// TwinCAT 3 PLC project PLC_OPEN_DRIVE
// Title: PlcOpenDrive
// Author: D.Hauer
// ProjectVersion: 00.50.3
// Description: MotionControl Achs Controller für externe Ansteuerung; NCI implementation
// ProgramVersion: 3.1.4022.4
// libraries:
//   Tc2_EtherCAT, * (Beckhoff Automation GmbH)
//   Tc2_MC2, * (Beckhoff Automation GmbH)
//   Tc2_MC2_Camming, * (Beckhoff Automation GmbH)
//   Tc2_MC2_Drive, * (Beckhoff Automation GmbH)
//   Tc2_NC, * (Beckhoff Automation GmbH)
//   Tc2_NCI, * (Beckhoff Automation GmbH)
//   Tc2_PlcInterpolation, * (Beckhoff Automation GmbH)
//   Tc2_Standard, * (Beckhoff Automation GmbH)
//   Tc2_System, * (Beckhoff Automation GmbH)
//   Tc2_Utilities, * (Beckhoff Automation GmbH)
//   Tc3_Module, * (Beckhoff Automation GmbH)
// project tree:
//   DOC/ DOCUMENTATION.TcPOU
//   DUTs/AXIS_CONTROL/ e_AxisFunction.TcDUT, ST_AxisController.TcDUT, ST_CamIn.TcDUT, ST_MotionOptions.TcDUT, ST_DataLog.TcDUT, ST_GearIn.TcDUT, ST_GearInMultiMaster.TcDUT, ST_Homing.TcDUT, ST_NcParam.TcDUT, ST_AxisStatusCompact.TcDUT, ST_In.TcDUT, ST_Out.TcDUT
//   DUTs/MAPPING/ U_AXIS_CTRL.TcDUT, U_AXIS_GEAR_IN.TcDUT, U_AXIS_GEAR_IN_MULTIMASTER.TcDUT, U_AXIS_HOMING.TcDUT, U_AXIS_INFO.TcDUT, U_AXIS_MOTION_OPTIONS.TcDUT, U_AXIS_NC_PARAMETER.TcDUT, U_AXIS_STATE.TcDUT
//   DUTs/MESSAGE/ e_Device.TcDUT, E_MessageType.TcDUT, e_Subdevice.TcDUT, ST_Message.TcDUT
//   DUTs/NC_AXIS/ E_AxisEncoderType.TcDUT, ST_AxisName.TcDUT, ST_BoolParam.TcDUT, ST_GearInParams.TcDUT, ST_GetCamInfoParams.TcDUT, ST_HaltParams.TcDUT, ST_HaltPhasingParams.TcDUT, ST_HomeParams.TcDUT, ST_JogParams.TcDUT, ST_MoveAbsParams.TcDUT, ST_MoveVeloParams.TcDUT, ST_Param.TcDUT, ST_PhasingAbsParams.TcDUT, ST_PhasingRelParams.TcDUT, ST_ReadParamParams.TcDUT, ST_StopParams.TcDUT, ST_WriteParamParams.TcDUT
//   / GlobalTextList.TcGTLO, PlcTask.TcTTO, Visualisierungsmanager.TcVMO (not stored)
//   GVLs/ GVL_AXIS_CTRL.TcGVL
//   POUs/Functions/ f_Builder.TcPOU, f_DelBit64.TcPOU, f_FolderDate.TcPOU, f_GetBit64.TcPOU, f_Len.TcPOU, f_Setbit64.TcPOU
//   POUs/ MAIN.TcPOU, NCI.TcPOU, P_CopleyWorkAround.TcPOU
//   POUs/MAPPING/ MAPPING_in.TcPOU, MAPPING_out.TcPOU
//   POUs/MSG/ fb_WriteData.TcPOU, f_MessageSet.TcPOU, p_Data.TcPOU, Visualization.TcVIS
//   POUs/NCI/ e_Ctrl_NciCommand.TcDUT, e_NciChannelError.TcDUT, E_NCI_INTERPRETER_STATE.TcDUT, FB_Ctrl_NciChannel.TcPOU, FB_NciChannel.TcPOU, GVL_NCI.TcGVL, I_NciChannel.TcIO, I_Nci_Ctrl.TcIO, ST_3D_Group.TcDUT, ST_CTRL_NCI.TcDUT, ST_Ctrl_NciMFuncCycle.TcDUT, ST_Index_Group.TcDUT, ST_Interface_Group.TcDUT, ST_NciChannel_Ref.TcDUT, ST_R_Parameter.TcDUT, ST_STATE_NCI.TcDUT
//   POUs/NC_AXIS/ FB_McPtpAxis.TcPOU, I_McAxis.TcIO
//   POUs/_FunctionBlocks/cam/ FB_CamIn_empty.TcPOU, fb_Camming.TcPOU, fb_Camming_Empty.TcPOU, FB_CamOut_Empty.TcPOU
//   POUs/_FunctionBlocks/ FB_AxisController.TcPOU, fb_Blink.TcPOU, fb_LocalTime.TcPOU, fb_ResetSercos.TcPOU, FB_XenaxEtherCATHoming.TcPOU

CONFIGURATION PLC_OPEN_DRIVE
    RESOURCE PLC ON TwinCAT3
        TASK PlcTask(INTERVAL := T#1ms, PRIORITY := 20);
        PROGRAM MAPPING_in WITH PlcTask : MAPPING_in;
        PROGRAM MAIN WITH PlcTask : MAIN;
        PROGRAM NCI WITH PlcTask : NCI;
        PROGRAM MAPPING_out WITH PlcTask : MAPPING_out;
    END_RESOURCE
END_CONFIGURATION

// ---- DUTs/AXIS_CONTROL/e_AxisFunction.TcDUT
{attribute 'to_string'}
TYPE e_AxisFunction :
(
  AXIS_DISABLE,
  AXIS_IDLE := 1,
  AXIS_ENABLE := 10,
  AXIS_HOME,
  AXIS_MOVE_POS,
  AXIS_MOVE_VELO,
  AXIS_RESET,
  AXIS_HALT,
  AXIS_STOP,

  // TODO: test
  AXIS_MOVE_BUFFER := 20,
  AXIS_MOVE_BUFFER_VELO,
  AXIS_WRITE_BUFFER_MODE,


  AXIS_PARAMETER   := 30, // axis function for reading and writing parameter


  AXIS_GEAR_IN    := 50,
  AXIS_GEAR_OUT,
  AXIS_GEAR_IN_MULTIMASTER,

  AXIS_CAM_IN   := 60,
  AXIS_CAM_OUT,
  AXIS_CAM_INFO,

  AXIS_SS1_STOP   :=  99,
  AXIS_BUSY       := 100,
  AXIS_ACK        := 300,
  AXIS_DONE       := 1000,

  ERROR           := 9000
)UINT;
END_TYPE

// ---- DUTs/AXIS_CONTROL/ST_AxisController.TcDUT
{attribute 'pack_mode' := '2'}
TYPE ST_AxisController :
STRUCT
  ToPlc    : ST_In;
  FromPlc  : ST_Out;
END_STRUCT
END_TYPE

// ---- DUTs/AXIS_CONTROL/ST_CamIn.TcDUT
TYPE ST_CamIn :
STRUCT
  MasterOffset      : REAL; 
  SlaveOffset       : REAL; 
  MasterScaling     : REAL;
  SlaveScaling      : REAL;

{IF defined (CAM)}
  {info 'CAMMING active'}
  StartMode         : Tc2_MC2_Camming.MC_StartMode;
  CamTableID        : Tc2_MC2_Camming.MC_CAM_ID;
{ELSE}
  StartMode         : INT;
  CamTableID        : UDINT;
{END_IF}

END_STRUCT
END_TYPE

// ---- DUTs/AXIS_CONTROL/ST_MotionOptions.TcDUT
TYPE ST_MotionOptions :
STRUCT
  eBufferMode   : Tc2_MC2.MC_BufferMode;

END_STRUCT
END_TYPE

// ---- DUTs/AXIS_CONTROL/ST_DataLog.TcDUT
TYPE ST_DataLog :
STRUCT
  WorkOrder : WORD;
  Duration  : REAL; // [ms]
  Position  : REAL;
END_STRUCT
END_TYPE

// ---- DUTs/AXIS_CONTROL/ST_GearIn.TcDUT
{attribute 'pack_mode' := '2'}
TYPE ST_GearIn :
STRUCT
  RatioNumerator  : REAL := 1.0; 
  RatioDenominator: UINT := 1; 
  Acceleration    : REAL;
  Deceleration    : REAL;
  Jerk            : REAL;
END_STRUCT
END_TYPE

// ---- DUTs/AXIS_CONTROL/ST_GearInMultiMaster.TcDUT
{attribute 'pack_mode' := '2'}
TYPE ST_GearInMultiMaster :
STRUCT  
  byAxisIDMaster1  : BYTE; // AxisID of Master1
  byAxisIDMaster2  : BYTE; // AxisID of Master2
  byAxisIDMaster3  : BYTE; // AxisID of Master3
  byAxisIDMaster4  : BYTE; // AxisID of Master4
  GearRatio1       : REAL; 
  GearRatio2       : REAL; 
  GearRatio3       : REAL; 
  GearRatio4       : REAL; 
  Acceleration     : REAL;
  Deceleration     : REAL;
  Jerk             : REAL;  
END_STRUCT
END_TYPE

// ---- DUTs/AXIS_CONTROL/ST_Homing.TcDUT
TYPE ST_Homing :
STRUCT
  bExecute      : BIT;

  stHomingParam : ST_HomeParams;
END_STRUCT
END_TYPE

// ---- DUTs/AXIS_CONTROL/ST_NcParam.TcDUT
TYPE ST_NcParam :
STRUCT
  bRead           : BIT;
  bWrite          : BIT;
  bValid          : BIT;

  (* reserve for future use *)
  // TwinCAT fills up to byte alignement, the declarations are not neccessarily required
  // for ease of use placeholders are hidden from intelli sense
  {attribute 'hide'}
  b3 : BIT;
  {attribute 'hide'}
  b4 : BIT;
  {attribute 'hide'}
  b5 : BIT;
  {attribute 'hide'}
  b6 : BIT;
  {attribute 'hide'}
  b7 : BIT;
  {attribute 'hide'}
  by1 : BYTE;

  ParameterNumber : Tc2_MC2.MC_AxisParameter;
  rValueWrite     : REAL; // value to write
  rValueRead      : REAL; // value from NC (Bools are cast to real)
END_STRUCT
END_TYPE

// ---- DUTs/AXIS_CONTROL/ST_AxisStatusCompact.TcDUT
{attribute 'pack_mode' := '2'}
TYPE ST_AxisStatusCompact :
STRUCT

    Error                : BIT;  (* axis error state *)

    (* PLCopen motion control statemachine states: *)
    ErrorStop            : BIT;
    Disabled             : BIT;
    Stopping             : BIT;

    StandStill           : BIT;
    DiscreteMotion       : BIT;
    ContinuousMotion     : BIT; 
    SynchronizedMotion   : BIT;

    Homing               : BIT;

    (* additional status - (PLCopen definition)*)
    ConstantVelocity     : BIT; 
    Accelerating         : BIT;
    Decelerating         : BIT;

    (* Axis.NcToPlc.StateDWord *)
    Operational          : BIT; 
    ControlLoopClosed    : BIT; (* operational and position control active *)
    HasJob               : BIT; 
    HasBeenStopped       : BIT; 
    NewTargetPosition    : BIT; (* new target position commanded during move *)
    InPositionArea       : BIT; 
    InTargetPosition     : BIT; 
 
    Homed                : BIT; 
    HomingBusy           : BIT; 
    MotionCommandsLocked : BIT; (* stop 'n hold *)
    SoftLimitMinExceeded : BIT; (* reverse soft travel limit exceeded *)
    SoftLimitMaxExceeded : BIT; (* forward soft travel limit exceeded *)

    Moving               : BIT; 
    PositiveDirection    : BIT; 
    NegativeDirection    : BIT; 
    NotMoving            : BIT; 
    Compensating         : BIT; (* superposition - overlayed motion *)

    ExtSetPointGenEnabled: BIT; 
    ExternalLatchValid   : BIT; 
    CamDataQueued        : BIT; 
    CamTableQueued       : BIT; 
    CamScalingPending    : BIT; 
    CmdBuffered          : BIT; 
    PTPmode              : BIT; 
    DriveDeviceError     : BIT; 
    IoDataInvalid        : BIT; 

    (* Axis.NcToPlc.CoupleState *)
    Coupled              : BIT;

END_STRUCT
END_TYPE

// ---- DUTs/AXIS_CONTROL/ST_In.TcDUT
{attribute 'pack_mode' := '2'}
TYPE ST_In :
STRUCT


  bFastStop         : BIT;  // Fast stop function of NC with mapped input

  {attribute 'hide'}
  b1 : BIT; // hide bit; for future use
  {attribute 'hide'}
  b2 : BIT; // hide bit; for future use
  {attribute 'hide'}
  b3 : BIT; // hide bit; for future use
  {attribute 'hide'}
  b4 : BIT; // hide bit; for future use
  {attribute 'hide'}
  b5 : BIT; // hide bit; for future use
  {attribute 'hide'}
  b6 : BIT;
  {attribute 'hide'}
  b7 : BIT;

  byAxisFuncPara    : BYTE; // additional parameter for Axis Function; e.g. used for AxisIndex on GearIn

  uiAxisFunctionReq : e_AxisFunction; // selected function for axis 

  (* LREAL required by process *)
  rSetPos           : LREAL;
  rSetVelo          : LREAL;
  rOverride         : LREAL;
  rAcc              : LREAL;
  rDec              : LREAL;
  iDirection        : INT;

  {attribute 'hide'}
  w1 : ARRAY[1..3] OF WORD;

END_STRUCT
END_TYPE

// ---- DUTs/AXIS_CONTROL/ST_Out.TcDUT
{attribute 'pack_mode' := '2'}
TYPE ST_Out :
STRUCT

  bEnabled    : BIT; // Enabled: check if ControlLoop is closed and active
  bReferenced : BIT; // Axis homing bit
  bReady      : BIT; // enabled & NOT bError & no Axis Function requested
  bBusy       : BIT; // axis function requested or active
  bError      : BIT;
  bTimeout    : BIT; // for move cmds or switching drive on timeout
  bInTarget   : BIT; // ActPos = SetPos --> position check is done with configured window in NC
  bStandstill : BIT; // No Error and NOT moving

  byAxisFuncPara      : BYTE; // mirror for additional parameter for Axis Function; e.g. used for AxisIndex on GearIn
  uiAxisFunctionState : e_AxisFunction; // mirror the requested axis function; 
                                        // +  100 = function busy; 
                                        // + 1000 = function done; 
                                        // + 9000 = function error
  uiErrorId           : UDINT;

  rActPos             : LREAL;
  rActVelo            : LREAL;
  rPosDiff            : LREAL;

  rSetPos             : LREAL;

  // HAUD
  // 2023 04 05
  dwCoupleState       : DWORD;   // cyclic information about axis couple state

  {attribute 'hide'}
  w1 : ARRAY[1..4] OF WORD;
END_STRUCT
END_TYPE

// ---- DUTs/MAPPING/U_AXIS_CTRL.TcDUT
TYPE U_AXIS_CTRL :
UNION

  stCtrl              : ARRAY[1..GVL_AXIS_CTRL.gciMaxAxis] OF ST_In;

{IF defined (AXIS_MAP)}
  {info 'U_AXIS_CTRL mapping activated'}
  byCtrl    AT %I*    : ARRAY[1..GVL_AXIS_CTRL.gciMaxAxis] OF
                        ARRAY[1..SIZEOF(ST_In)] OF BYTE;
{ELSE}
  byCtrl              : ARRAY[1..GVL_AXIS_CTRL.gciMaxAxis] OF
                        ARRAY[1..SIZEOF(ST_In)] OF BYTE;
{END_IF}
END_UNION
END_TYPE

// ---- DUTs/MAPPING/U_AXIS_GEAR_IN.TcDUT
TYPE U_AXIS_GEAR_IN :
UNION

  stCtrl              : ARRAY[1..GVL_AXIS_CTRL.gciMaxAxis] OF ST_GearIn;

{IF defined (AXIS_MAP)}
  {info 'U_AXIS_GEAR_IN mapping activated'}
  byCtrl    AT %I*    : ARRAY[1..GVL_AXIS_CTRL.gciMaxAxis] OF
                        ARRAY[1..SIZEOF(ST_GearIn)] OF BYTE;
{ELSE}
  byCtrl              : ARRAY[1..GVL_AXIS_CTRL.gciMaxAxis] OF
                        ARRAY[1..SIZEOF(ST_GearIn)] OF BYTE;
{END_IF}
END_UNION
END_TYPE

// ---- DUTs/MAPPING/U_AXIS_GEAR_IN_MULTIMASTER.TcDUT
TYPE U_AXIS_GEAR_IN_MULTIMASTER :
UNION

  stCtrl              : ARRAY[1..GVL_AXIS_CTRL.gciMaxAxis] OF ST_GearInMultiMaster;

{IF defined (AXIS_MAP)}
  {info 'U_AXIS_GEAR_IN mapping activated'}
  byCtrl    AT %I*    : ARRAY[1..GVL_AXIS_CTRL.gciMaxAxis] OF
                        ARRAY[1..SIZEOF(ST_GearInMultiMaster)] OF BYTE;
{ELSE}
  byCtrl              : ARRAY[1..GVL_AXIS_CTRL.gciMaxAxis] OF
                        ARRAY[1..SIZEOF(ST_GearInMultiMaster)] OF BYTE;
{END_IF}
END_UNION
END_TYPE

// ---- DUTs/MAPPING/U_AXIS_HOMING.TcDUT
TYPE U_AXIS_HOMING :
UNION

  stCtrl              : ARRAY[1..GVL_AXIS_CTRL.gciMaxAxis] OF ST_Homing;

{IF defined (AXIS_MAP)}
  {info 'U_AXIS_HOMING mapping activated'}
  byCtrl    AT %I*    : ARRAY[1..GVL_AXIS_CTRL.gciMaxAxis] OF
                        ARRAY[1..SIZEOF(ST_Homing)] OF BYTE;
{ELSE}
  byCtrl              : ARRAY[1..GVL_AXIS_CTRL.gciMaxAxis] OF
                        ARRAY[1..SIZEOF(ST_Homing)] OF BYTE;
{END_IF}
END_UNION
END_TYPE

// ---- DUTs/MAPPING/U_AXIS_INFO.TcDUT
TYPE U_AXIS_INFO :
UNION

  stState             : ARRAY[1..GVL_AXIS_CTRL.gciMaxAxis] OF ST_AxisStatusCompact;

{IF defined (AXIS_MAP)}
  {info 'U_AXIS_INFO mapping activated'}
  byState  AT %Q*     : ARRAY[1..GVL_AXIS_CTRL.gciMaxAxis] OF
                        ARRAY[1..SIZEOF(ST_AxisStatusCompact)] OF BYTE;
{ELSE}
  byState             : ARRAY[1..GVL_AXIS_CTRL.gciMaxAxis] OF
                        ARRAY[1..SIZEOF(ST_AxisStatusCompact)] OF BYTE;
{END_IF}
END_UNION
END_TYPE

// ---- DUTs/MAPPING/U_AXIS_MOTION_OPTIONS.TcDUT
TYPE U_AXIS_MOTION_OPTIONS :
UNION

  stCtrl              : ARRAY[1..GVL_AXIS_CTRL.gciMaxAxis] OF ST_MotionOptions;

{IF defined (AXIS_MAP)}
  {info 'U_AXIS_MOTION_OPTIONS mapping activated'}
  byCtrl    AT %I*    : ARRAY[1..GVL_AXIS_CTRL.gciMaxAxis] OF
                        ARRAY[1..SIZEOF(ST_MotionOptions)] OF BYTE;
{ELSE}
  byCtrl              : ARRAY[1..GVL_AXIS_CTRL.gciMaxAxis] OF
                        ARRAY[1..SIZEOF(ST_MotionOptions)] OF BYTE;
{END_IF}
END_UNION
END_TYPE

// ---- DUTs/MAPPING/U_AXIS_NC_PARAMETER.TcDUT
TYPE U_AXIS_NC_PARAMETER :
UNION

  stState             : ARRAY[1..GVL_AXIS_CTRL.gciMaxAxis] OF ST_NcParam;

{IF defined (AXIS_MAP)}
  {info 'U_AXIS_NC_PARAM mapping activated'}
  byState   AT %Q*    : ARRAY[1..GVL_AXIS_CTRL.gciMaxAxis] OF
                        ARRAY[1..SIZEOF(ST_NcParam)] OF BYTE;
{ELSE}
  byState             : ARRAY[1..GVL_AXIS_CTRL.gciMaxAxis] OF
                        ARRAY[1..SIZEOF(ST_NcParam)] OF BYTE;
{END_IF}
END_UNION
END_TYPE

// ---- DUTs/MAPPING/U_AXIS_STATE.TcDUT
TYPE U_AXIS_STATE :
UNION

  stState             : ARRAY[1..GVL_AXIS_CTRL.gciMaxAxis] OF ST_Out;

{IF defined (AXIS_MAP)}
  {info 'U_AXIS_STATE mapping activated'}
  byState   AT %Q*    : ARRAY[1..GVL_AXIS_CTRL.gciMaxAxis] OF
                        ARRAY[1..SIZEOF(ST_Out)] OF BYTE;
{ELSE}
  byState             : ARRAY[1..GVL_AXIS_CTRL.gciMaxAxis] OF
                        ARRAY[1..SIZEOF(ST_Out)] OF BYTE;
{END_IF}
END_UNION
END_TYPE

// ---- DUTs/MESSAGE/e_Device.TcDUT
{attribute 'to_string'}
TYPE e_Device :
(
  General         := 0,

  // first NC Axis, all other Axis are incremented
  Axis            := 1000,

  // NCI channel control instance
  NciChannelCtrl  := 2000,

  // NCI channel
  NciChannel      := 3000,

  // message function blocks
  Data            := 10000
)DINT;
END_TYPE

// ---- DUTs/MESSAGE/E_MessageType.TcDUT
{attribute 'strict'}
{attribute 'to_string'}
TYPE E_MessageType :
(
  eMessageEmpty,
  eMessageInfo,
  eMessageWarn,
  eMessageError
)DINT;
END_TYPE

// ---- DUTs/MESSAGE/e_Subdevice.TcDUT
{attribute 'strict'}
{attribute 'to_string'}
TYPE e_Subdevice :
(
  // sub device for message system
  General := 0,
  // Motion Control FB Instances
  fbPower,
  fbReset,
  fbResetSercos,
  fbHalt,
  fbStop,
  fbHome,
  fbJog,
  fbMoveVelocity1,
  fbMoveVelocity2,
  fbMoveAbsolute1,
  fbMoveAbsolute2,
  fbMoveEndless,
  fbMovePtP,

  fbGearIn := 50,
  fbGearOut,
  fbGearInMultiMaster,

  fbCamIn := 60,
  fbCamOut,

  fbReadParameter := 100,
  fbReadBoolParameter,
  fbWriteParameter,
  fbWriteBoolParameter,

	fbBuildGroup := 200,
	fbClearGroup,
	fbLoadProg,
	fbResetItp,
	fbStartStopItp,
	fbEStopItp,
	fbStepOnAfterEStopItp,
	fbConfirmHskItp,
	fbDelDtgItp,
	fbNciFeedTablePreparation,
	fbNciFeedTable,
	fbReadLine,
  fbItpReadRParams,
  fbItpWriteRParams,

  Get_ItpState,
  Get_Error,

  AxisMode      := 1000,

  Ctrl_Nci_Cmd  := 2000
)DINT;
END_TYPE

// ---- DUTs/MESSAGE/ST_Message.TcDUT
TYPE ST_Message :
STRUCT
  eType         : e_MessageType;
  eDevice       : e_Device;
  eSubdevice    : e_SubDevice;
  {attribute 'displaymode':='hex'}
  iErrorNumber  : LINT;
  tTime         : STRING(24);
  sText         : STRING(256);
END_STRUCT
END_TYPE

// ---- DUTs/NC_AXIS/E_AxisEncoderType.TcDUT
{attribute 'to_string'}
TYPE E_AxisEncoderType :
(
  NoEncoder := 0,
  
  Simulation_Encoder,
  
  M3000_Enc,
  M31x0_M2000_Enc,
  MDP_511_Enc,
  MDP_500_501_Enc,
  MDP_510_Enc,
  KL30xx_Enc,
  SERCOS_EtherCAT_SoE_Pos,
  SERCOS_EtherCAT_SoE_Pos_Velo,
  Binary_Enc,
  M2510_Enc,
  FOX50_Enc                     := 12,
  AX2000_Lightbus               := 14,
  Provi_DriveMC_Simodrive_611U,
  Universal_Encoder_varBitmask,
  NC_Backplane,
  spec_CANopen_Typ,
  MDP_513_DS402,
  AX2xx_B900,
  KL5151_Encoder                := 21,
  IP5209_Encoder                := 24,
  KL2531_KL2541_Encoder,
  KL2532_KL2542_Encoder,
  Time_Base_Encoder,
  TCom_Encoder_SoftDrive
)UDINT;
END_TYPE

// ---- DUTs/NC_AXIS/ST_AxisName.TcDUT
TYPE ST_AxisName :
STRUCT
  sName     : STRING(31);
  bValid    : BOOL;
END_STRUCT
END_TYPE

// ---- DUTs/NC_AXIS/ST_BoolParam.TcDUT
TYPE ST_BoolParam :
STRUCT
  bValue      : BOOL;
  bValid      : BOOL;
  bWriteToNc  : BOOL;
END_STRUCT
END_TYPE

// ---- DUTs/NC_AXIS/ST_GearInParams.TcDUT
TYPE ST_GearInParams :
STRUCT
  Enable        : BOOL;
  GearRatio     : LREAL;
  GearRatio2    : LREAL;
  GearRatio3    : LREAL;
  GearRatio4    : LREAL;
  Acceleration  : LREAL;
  Deceleration  : LREAL;
  Jerk          : LREAL;
  Options       : Tc2_MC2.ST_GearInMultiMasterOptions;
END_STRUCT
END_TYPE

// ---- DUTs/NC_AXIS/ST_GetCamInfoParams.TcDUT
TYPE ST_GetCamInfoParams :
STRUCT
  AtMasterPosition  : BOOL;
  MasterPosition    : LREAL;
END_STRUCT
END_TYPE

// ---- DUTs/NC_AXIS/ST_HaltParams.TcDUT
TYPE ST_HaltParams :
STRUCT
  Deceleration  : LREAL;
  Jerk          : LREAL;
  BufferMode    : Tc2_MC2.MC_BufferMode;
END_STRUCT
END_TYPE

// ---- DUTs/NC_AXIS/ST_HaltPhasingParams.TcDUT
TYPE ST_HaltPhasingParams :
STRUCT
  Deceleration  : LREAL;
  Jerk          : LREAL;
END_STRUCT
END_TYPE

// ---- DUTs/NC_AXIS/ST_HomeParams.TcDUT
TYPE ST_HomeParams :
STRUCT
  Position              : LREAL;
  HomingMode            : Tc2_MC2.MC_HomingMode;
  Options               : Tc2_MC2.ST_HomingOptions;
  InvertHomeSensor      : BIT := FALSE;   //Set to true, if the home sensor is normally closed.
  SimulateHomeSensor    : BIT := FALSE;   //Set to true, if the axis should be homed on encoder index only. The homing methode 'hardware sync' must be used then.
  UseLimitMin           : BIT := TRUE;    //Set to false, if there is no negative limit sensor.
  InvertLimitMin        : BIT := FALSE;   //Set to true, if the negative limit sensor is normally closed.
  HomeOnLimitMin        : BIT := FALSE;   //Set to true, if the negative limit sensor should be used for homing. 
  UseLimitMax           : BIT := TRUE;    //Set to false, if there is no positive limit sensor.
  InvertLimitMax        : BIT := FALSE;   //Set to true, if the positive limit sensor is normally closed.
  HomeOnLimitMax        : BIT := FALSE;   //Set to true, if the positive limit sensor should be used for homing. 
  
  // It is not allowed to use more than 1 of the 3 switches: SimulateHomeSensor, HomeOnLimitMin, HomeOnLimitMax
  
END_STRUCT
END_TYPE

// ---- DUTs/NC_AXIS/ST_JogParams.TcDUT
TYPE ST_JogParams :
STRUCT
  JogForward    : BOOL;
  JogBackwards  : BOOL;
  Mode          : Tc2_MC2.E_JogMode;
  Position      : LREAL;
  Velocity      : LREAL;
  Acceleration  : LREAL;
  Deceleration  : LREAL;
  Jerk          : LREAL;
END_STRUCT
END_TYPE

// ---- DUTs/NC_AXIS/ST_MoveAbsParams.TcDUT
TYPE ST_MoveAbsParams :
STRUCT
	Position		: LREAL;
	Velocity		: LREAL;
	Acceleration	: LREAL;
	Deceleration	: LREAL;
	Jerk			: LREAL;
	BufferMode		: Tc2_MC2.MC_BufferMode;
END_STRUCT
END_TYPE

// ---- DUTs/NC_AXIS/ST_MoveVeloParams.TcDUT
TYPE ST_MoveVeloParams :
STRUCT
  Velocity      : LREAL;
  Acceleration  : LREAL;
  Deceleration  : LREAL;
  Jerk          : LREAL;
  Direction     : Tc2_MC2.MC_Direction := MC_Positive_Direction;
  BufferMode    : Tc2_MC2.MC_BufferMode;
END_STRUCT
END_TYPE

// ---- DUTs/NC_AXIS/ST_Param.TcDUT
TYPE ST_Param :
STRUCT
  fValue    : LREAL;
  bValid    : BOOL;
  bWriteToNc  : BOOL;
END_STRUCT
END_TYPE

// ---- DUTs/NC_AXIS/ST_PhasingAbsParams.TcDUT
TYPE ST_PhasingAbsParams :
STRUCT
	PhaseShift		: LREAL;
	Velocity		: LREAL;
	Acceleration	: LREAL;
	Deceleration	: LREAL;
	Jerk			: LREAL;
END_STRUCT
END_TYPE

// ---- DUTs/NC_AXIS/ST_PhasingRelParams.TcDUT
TYPE ST_PhasingRelParams :
STRUCT
	PhaseShift		: LREAL;
	Velocity		: LREAL;
	Acceleration	: LREAL;
	Deceleration	: LREAL;
	Jerk			: LREAL;
END_STRUCT
END_TYPE

// ---- DUTs/NC_AXIS/ST_ReadParamParams.TcDUT
TYPE ST_ReadParamParams :
STRUCT
	ParameterNumber	: Tc2_MC2.MC_AxisParameter;
END_STRUCT
END_TYPE

// ---- DUTs/NC_AXIS/ST_StopParams.TcDUT
TYPE ST_StopParams :
STRUCT
	Deceleration	: LREAL;
	Jerk			: LREAL;
END_STRUCT
END_TYPE

// ---- DUTs/NC_AXIS/ST_WriteParamParams.TcDUT
TYPE ST_WriteParamParams :
STRUCT
  ParameterNumber : Tc2_MC2.MC_AxisParameter;
  Value           : LREAL;
END_STRUCT
END_TYPE

// ---- POUs/NCI/e_Ctrl_NciCommand.TcDUT
{attribute 'qualified_only'}
{attribute 'to_string'}
TYPE e_Ctrl_NciCommand :
(
  NO_NCI            := -10,
  NO_AXIS_GROUP     := -2,
  NO_AXIS_INDEX     := -1,
  NO_INIT,
  INIT,
  IDLE,
  RESET,
  LOAD_PROG,
  FEED_TABLE,
  BUILD_GROUP,
  CLEAR_GROUP,

  START         := 10,
  STOP,
  STO_STOP,
  RESTART_STEP_ON,

  M_FUNC_QUIT   := 20,

  READ_R_PARA   := 30,
  WRITE_R_PARA  := 40,

  CMD_BUSY      := 100,
  CMD_DONE      := 1000,
  CMD_ERROR     := 9000
)DINT;
END_TYPE

// ---- POUs/NCI/e_NciChannelError.TcDUT
{attribute 'qualified_only'}
{attribute 'strict'}
TYPE e_NciChannelError :
(
  e_Null,
  e_InvalidReference_ChannelRef,
  e_AxisConfigurationMismatch_McAxis,
  e_AxisConfigurationMismatch_AuxAxis


);
END_TYPE

// ---- POUs/NCI/E_NCI_INTERPRETER_STATE.TcDUT
// Interpreter state, see also library tc2_nci.Global_Variables.NCI_INTERPRETER_xxx
//  Date    Name  Version   Remarks
//  2016/09/29  FJK   1.0     1st Version
{attribute -'to_string'}
TYPE E_NCI_INTERPRETER_STATE :
(
  NCI_INTERPRETER_INITFAILED := 0,
  NCI_INTERPRETER_IDLE := 1,
  NCI_INTERPRETER_READY := 2,
  NCI_INTERPRETER_STARTED := 3,
  NCI_INTERPRETER_SCANNING := 4,
  NCI_INTERPRETER_RUNNING := 5,
  NCI_INTERPRETER_STAY_RUNNING := 6,
  NCI_INTERPRETER_WRITETABLE := 7,
  NCI_INTERPRETER_SEARCHLINE := 8,
  NCI_INTERPRETER_END := 9,
  NCI_INTERPRETER_SINGLESTOP := 10, 
  NCI_INTERPRETER_ABORTING := 11,
  NCI_INTERPRETER_ABORTED := 12,
  NCI_INTERPRETER_FAULT := 13,
  NCI_INTERPRETER_RESET := 14,
  NCI_INTERPRETER_STOP := 15,
  NCI_INTERPRETER_WAITFUNC := 16,
  NCI_INTERPRETER_FLUSHBUFFERS := 17
) DWORD;    //Basis-Datentyp
END_TYPE

// ---- POUs/NCI/ST_3D_Group.TcDUT
{attribute 'pack_mode' := '2'}
TYPE ST_3D_Group :
STRUCT
  nXAxisId    : UDINT := 1;
  nYAxisId    : UDINT := 2;
  nZAxisId    : UDINT := 3;
  nQ1AxisId   : UDINT;
  nQ2AxisId   : UDINT;
  nQ3AxisId   : UDINT;
  nQ4AxisId   : UDINT;
  nQ5AxisId   : UDINT;
END_STRUCT
END_TYPE

// ---- POUs/NCI/ST_CTRL_NCI.TcDUT
{attribute 'pack_mode' := '2'}
TYPE ST_CTRL_NCI :
STRUCT
  eCmd        : e_Ctrl_NciCommand := e_Ctrl_NciCommand.INIT;
  rOverride   : REAL := 47.11;

END_STRUCT
END_TYPE

// ---- POUs/NCI/ST_Ctrl_NciMFuncCycle.TcDUT
{attribute 'pack_mode' := '2'}
TYPE ST_Ctrl_NciMFuncCycle :
STRUCT
  FastMFuncMask   : ARRAY [1..5] OF DWORD;
  HskMFuncNo      : UINT;
  HskMFuncReq     : WORD;
  HFuncValue      : UDINT; 
END_STRUCT
END_TYPE

// ---- POUs/NCI/ST_Index_Group.TcDUT
{attribute 'pack_mode' := '2'}
TYPE ST_Index_Group :
STRUCT
  nXAxisIdx     : UDINT := 1;
  nYAxisIdx     : UDINT := 2;
  nZAxisIdx     : UDINT := 3;

  nQ1AxisIdx    : UDINT;
  nQ2AxisIdx    : UDINT;
  nQ3AxisIdx    : UDINT;
  nQ4AxisIdx    : UDINT;
  nQ5AxisIdx    : UDINT;
END_STRUCT
END_TYPE

// ---- POUs/NCI/ST_Interface_Group.TcDUT
{attribute 'pack_mode' := '2'}
TYPE ST_Interface_Group :
STRUCT
  I_Idx_XAxis     : I_McAxis;
  I_Idx_YAxis     : I_McAxis;
  I_Idx_ZAxis     : I_McAxis;

  I_Idx_Q1Axis    : I_McAxis;
  I_Idx_Q2Axis    : I_McAxis;
  I_Idx_Q3Axis    : I_McAxis;
  I_Idx_Q4Axis    : I_McAxis;
  I_Idx_Q5Axis    : I_McAxis;
END_STRUCT
END_TYPE

// ---- POUs/NCI/ST_NciChannel_Ref.TcDUT
TYPE ST_NciChannel_Ref :
STRUCT
  NcToPlc AT %I*: NcToPlc_NciChannel_Ref;   //  Externer Datentyp!
  PlcToNc AT %Q*: PlcToNc_NciChannel_Ref;   //  Externer Datentyp!
END_STRUCT
END_TYPE

// ---- POUs/NCI/ST_R_Parameter.TcDUT
{attribute 'pack_mode' := '2'}
TYPE ST_R_Parameter :
STRUCT
{IF defined (AXIS_MAP)}
  {info 'NCI channel mapping for test'}
  _nStart        AT %I* : DINT;
  _nCount        AT %I* : DINT;
  _rRParamsWrite AT %I* : ARRAY[0..GVL_NCI.cRParamCount] OF LREAL;
  _rRParamsRead  AT %Q* : ARRAY[0..GVL_NCI.cRParamCount] OF LREAL;
{ELSE}
  _nStart               : DINT := 901;
  _nCount               : DINT :=   4;
  _rRParamsWrite        : ARRAY[0..GVL_NCI.cRParamCount] OF LREAL := [11.11, 22.22, 33.33, 456.22];
  _rRParamsRead         : ARRAY[0..GVL_NCI.cRParamCount] OF LREAL;
{END_IF}
END_STRUCT
END_TYPE

// ---- POUs/NCI/ST_STATE_NCI.TcDUT
{attribute 'pack_mode' := '2'}
TYPE ST_STATE_NCI :
STRUCT
  eState        : e_Ctrl_NciCommand; // eCmd with offsets for busy and done

  bMFuncReq     : BIT;  // M function request is active from channel

  nMFunc        : WORD; // number of active M function

  nItpState     : UINT; 
                         (*  Interpreter Operation State:
                            0  = Init failed
                            1  = Idle
                            2  = Ready
                            3  = Started
                            4  = Scanning
                            5  = Running
                            6  = Stay running
                            7  = Write table
                            8  = Search line
                            9  = End
                            10 = Single Step
                            11 = Aborting
                            12 = Aborted
                            13 = Fault
                            14 = Reset
                            15 = Stop
                            16 = Wait function
                            17 = Flush buffers
                          *) 

  rAxisOverride : REAL; // active override in cyclic NCI interface

END_STRUCT
END_TYPE

// ---- GVLs/GVL_AXIS_CTRL.TcGVL
{attribute 'qualified_only'}
VAR_GLOBAL CONSTANT

{IF defined (WIN)}
  {info 'WIN folders'}
  gcsLogDir         : STRING := 'C:\TwinCAT\#MsgFiles\';
{ELSE}
  {info 'BSD folders'}
  gcsLogDir         : STRING := '/usr/local/etc/TwinCAT/#MsgFiles/';
{END_IF}

  gcsLogFile        : STRING := 'Msg_PlcOpenDrive_';

  gciMaxMessage     : INT := 200; // max entry in message list
  gciMaxAxis        : INT :=  3;

{IF defined (CAM)}
  {info 'camming active'}
  cCam                  : BOOL := TRUE;
{ELSE}
  {info 'camming NOT active'}
  cCam                  : BOOL := FALSE;
{END_IF}

  
//V 00.07
//04.11.2021
//HauD
// GearIn, GearOut added

// V 00.08
//24.03.2022
//HauD
// simple ptp movement with only one instance of MC functionblock
// file writing for logging now globally enable/disable
// intern message list is always used
// ref in property deleted
// axis pointer is used


// V 00.09
// 25.03.2022
// HAUD
// parameter handling changed
// NULL initialization of methods implemented

// V 00.10 - V 00.11
// 29.03.2022
// HAUD
// TEST

// V 00.12
// 29.03.2022
// HAUD
// Merge TEST and server version
// Visu page for message diag
// OP state before ADS READ on NC Axis
// INIT logging at startup
// enum to_string with use of 4024 compiler

// V 00.13
// 14.04.2022
// CamIn and CamOut added
// Changed Compiler Version to 3.1.4024.0. This is needed to enable conditional pragmas

// V 00.14
// 03.06.2022
// GearInMultiMaster added

// V 00.15
// 29.06.2022
// HAUD
// defines deleted, defines in code do not work, therefore all defines for camming deleted
// stop method in FB_McPtPAxis added.

// V00.16
// 30.06..2022
// HAUD
// FB_AxisController, code refactoring
//    Axis function states are now calling corresponding actions to improve readability
// SS1 stop with static check (SEL)

// V00.17
// 18.07.2022
// HAUD
// CAM_OUT now with FB check instead of mapping check

// V00.18
// 19.07.2022
// Axis startup, changes according to test
// ADS communication to AxisName changed, ADS Err 1796

// V00.19
// 27.07.2022
// HAUD
// Axis startup expanded to Encodertype for automatic Sercos selection
// fb_AxisController.bSercosAxis changed from input to output var
// CamOut checked with logging for couple state

// V00.20
// 27.07.2022
// HAUD
// Axis startup AdsRead.ERR automatic re-startup

// V00.21
// 06.10.2022
// HAUD
// test case for MOVE_VELO; HALT
// Halt() with standstill check
// MOVE_VELO, fbMoveEndless.Position feed check
// AXIS_HALT, standstill control with timeout and RESET
// AXIS_MOVE_BUFFER_VELO, two instances changing velocity during function execution, if required velo is reached, done OR keep function alive and change to velo2 and wait for done


// V00.22
// 13.10.2022
// HAUD
// AXIS_HALT standstill check changed to NotMoving

// V00.23
// 14.10.2022
// HAUD
// AXIS_MOVE_VELO - chsnged to MC_Velocity; Ctrl.iDirection is evaluated, 1 - positive; 3 - negative

// V00.24
// 15.10.2022
// HAUD
// code revision from testing
// Compiler def TEST      - TwinSAFE Alias device muted
// Compiler def AXIS_MAP  - cyclic mapping ST_AxisController
// Compiler def WIN       - windows file names for logging

// V00.25
// 15.10.2022
// HAUD
// Compiler def CAM      - contitional activation of camming lib
// MC_Camming lib now optional

// V00.26
// 16.10.2022
// HAUD
// cam folder missing, added by push
// property of MC2_Camming.lib is set to optional
// Compiler def:  - TEST      [forces SafetyOK internally]
//                - AXIS_MAP  [ST_AxisController will be mapped variable --> connection to second TEST_PLC]
//                - WIN       [windows file names are used]
//                - CAM       [MC2_Camming.lib is active --> if entry is not present, empty FBs are used]

// V00.27
// 19.10.2022
// HAUD
// R/W of axis parameter now possible without safety bit from Alias Device

// V00.28
// 20.10.2022
// HAUD
// GearOut and Disable are available during safety off.

// V00.30
// 23.10.2022
// HAUD
// NCI implementation of for basic use with g-Code files

// V00.32
// 25.10.2022
// HAUD
// consistent Datatypes for NCI define

// V00.33
// 25.10.2022
// HAUD
// NCI() call added to TaskReference
// NCI() works the ADS interface
// cyclic interface for NCI channels as global data structs
// plausibility checks

// V00.34
// 25.10.2022
// HAUD
// compiler defines test

// V00.35
// 25.10.2022
// HAUD
// BUG fb_AxisController.bSS1 state bereinigt

// V00.36
// 25.10.2022
// HAUD
// defines for test cases with mapping to extern plc
// 

// V00.37
// 25.10.2022
// HAUD
// defines for test cases with mapping to extern plc
// properties in fb_Ctrl_NciChannel are now using fb Instance of FB_NciChannel
// R Parameter window limited to 10

// V00.38
// 25.10.2022
// HAUD
// testing

// V00.39
// 31.10.2022
// HAUD
// quit of M function now on cyclic interface
// new member in ST_STATE_NCI  .ItpState - Interpreter state from cyclic NCI channel interfacwe 

// V00.40
// 02.11.2022
// HAUD
// testing

// V00.41
// 18.01.2023
// - BufferMode switch for e_AxisFunction.AXIS_MOVE_BUFFER and AXIS_MOVE_BUFFER_VELO

// V00.42
// HAUD
// 14.03.2023
// CAM_OUT check changed to strict eval

// V00.43
// HAUD
// 17.03.2023
// MC_BufferModes, additional error check in FB_McPtpAxis added (MoveAbsolute 1&2)

// V00.44
// HAUD
// 17.03.2023
// code review for missing stState.uiErrorId information to extern

// V00.45
// HAUD
// 27.03.2023
// debug for missing stState.uiErrorId information to extern
//
// 31.03.2023
// Axis_Cam_Out; ignore fb_CamOut error, retry if still coupled

// V00.46
// HAUD
// 05.04.2023
// Axis_Cam_Out; ignore axis function if not coupled
// fbAxis.pAxisRef^.NcToPlc.CoupleState added to ST_OUT

// V00.47
// HAUD
// 27.04.2023
// draft for redesign Camming lib implementation
// fb_CamIn_V2 replaces fb_CamIn

// V00.48 new branch on git server
// HAUD
// 26.05.2023
// ST_In; ST_Out change REAL --> LREAL

// V00.48.01
// HAUD
// 17.10.2023
// more than 100 Axis declared in project --> ADS handles can not be created for all axis, StartUp FB_McPtpAxis stopps with error, manual reset required --> changed to closer monitoring and retry
// FB_McPtpAxis.StartupError    - added if ADS Read error, StartUp error state wait for Reset
// FB_McPtpAxis.ErrorReset      - added StartUp error state reset (restarts StartUp state machine)
// FB_AxisController.Axis_Init  - state machine is checked for fbAxis.StartUpError, automatic axis reset and retry

// V00.50.1
// HAUD
// 19.10.2023
// CAMMING implementation with table manipulation
// redesign for modular use --> FB_AxisController does not host camming lib
// interface implementation for downward compatibility

// V00.48.93
// HAUD
// 15.02.2024
// Buffered moves with additional info on ST_Out.rSetPos

// V00.50.2
// HAUD
// 07.03.2024
// merge changes from field V 00.48.95
// buffered move
// message handling

// V00.50.3
// HAUD
// 11.03.2024
// AXIS_MAP pragma through dedicated PRG (in/out)



  Version           : STRING := 'V 00.50.3';
END_VAR
VAR_GLOBAL

  gfbAxisController : ARRAY[1..gciMaxAxis] OF FB_AxisController;  // cyclic interface for accepting and executing orders
  gstAxisControl    : ARRAY[1..gciMaxAxis] OF ST_AxisController;  // structure for cyclic interface


  gstAxisParam                  : ARRAY[1..gciMaxAxis] OF ST_NcParam;         // R/W struct for a single parameter
  gstHomeParam                  : ARRAY[1..gciMaxAxis] OF ST_HomeParams;      // homing parameter for each axis

  gstAxisCamParam               : ARRAY[1..gciMaxAxis] OF ST_CamIn;
  gstAxisGearParam              : ARRAY[1..gciMaxAxis] OF ST_GearIn;
  gstAxisGearMultiMasterParam   : ARRAY[1..gciMaxAxis] OF ST_GearInMultiMaster;

  gstMotionOptions              : ARRAY[1..gciMaxAxis] OF ST_MotionOptions;

  // diag data
  gbyAxisIdxGearIn              : ARRAY[1..gciMaxAxis]      OF BYTE; // diag for Axis gear in
  
  gbyAxisIdxGearInMultiMaster   : ARRAY[1..gciMaxAxis,1..4] OF BYTE; // diag for Axis gear in multi master
  
  gbyAxisIdxCamIn               : ARRAY[1..gciMaxAxis]      OF BYTE; // diag for Axis cam in

  gatMessages       : ARRAY[1..gciMaxMessage] OF ST_Message;
  giMsgIndex        : INT := 1;
  giErrorIndex      : INT := 0;

  gfbLocalTime      : fb_LocalTime;
  gdtLocalTime      : DT;
  gsLocalTime       : STRING;

{IF defined (AXIS_MAP)}
  {info 'TEST ST_AxisController'}
  gbEnableLogging   : BOOL := TRUE;
{ELSE}
  gbEnableLogging   : BOOL;
{END_IF}
END_VAR

// ---- POUs/NCI/GVL_NCI.TcGVL
{attribute 'qualified_only'}
VAR_GLOBAL CONSTANT
  cPathSteps            : UINT    := 5;  //Path-Steps[0]:Velo, [1]:X, [2]:Y, [3]:Z
  cMcAxisCount          : UINT    := 8;
  cAuxAxisCount         : UINT    := 8;
  cRParamCount          : UINT    := 10;

  cNciSpec              : STRING  := 'NCI_Spec_Ch_';

  cMaxNciCh             : INT     :=  1;

{IF defined (NCI)}
  {info 'NCI channel active'}
  cNci                  : BOOL := TRUE;
{ELSE}
  {info 'NCI channel NOT active'}
  cNci                  : BOOL := FALSE;
{END_IF}


{IF defined (WIN)}
  {info 'WIN folders'}
  cNciDir              : STRING   := 'C:\TwinCAT\Mc\Nci\';
{ELSE}
  {info 'BSD folders'}
  cNciDir              : STRING   := '/usr/local/etc/TwinCAT/Mc/Nci/';
{END_IF}
END_VAR
VAR_GLOBAL

{IF defined (AXIS_MAP)}
  {info 'NCI channel mapping for test'}
  gstAxisIndex      AT %I*    : ARRAY[1..cMaxNciCh] OF ST_Index_Group;  // index of gstAxisCtontrl[]
  gstAxisConfig     AT %I*    : ARRAY[1..cMaxNciCh] OF ST_3D_Group;     // NC Axis Id to build NCI group

  gstChannelCtrl    AT %I*    : ARRAY[1..cMaxNciCh] OF ST_CTRL_NCI;
  gstChannelState   AT %Q*    : ARRAY[1..cMaxNciCh] OF ST_STATE_NCI;

  gsProgName        AT %I*    : ARRAY[1..cMaxNciCh] OF STRING(255);
  gsProgNameActive  AT %Q*    : ARRAY[1..cMaxNciCh] OF STRING(255);
{ELSE}

  // ADS R/W data:
  gstAxisIndex                : ARRAY[1..cMaxNciCh] OF ST_Index_Group;  // index of gstAxisCtontrl[]
  gstAxisConfig               : ARRAY[1..cMaxNciCh] OF ST_3D_Group;     // NC Axis Id to build NCI group

  gstChannelCtrl              : ARRAY[1..cMaxNciCh] OF ST_CTRL_NCI;
  gstChannelState             : ARRAY[1..cMaxNciCh] OF ST_STATE_NCI;

  gsProgName                  : ARRAY[1..cMaxNciCh] OF STRING(255):= ['/usr/local/etc/TwinCAT/Mc/Nci/Test_GST.nc'];
  gsProgNameActive            : ARRAY[1..cMaxNciCh] OF STRING(255);
{END_IF}

  gstRParameter               : ARRAY[1..cMaxNciCh] OF ST_R_Parameter;

{IF defined (NCI)}
  gfbNciCtrl            : ARRAY[1..cMaxNciCh] OF FB_Ctrl_NciChannel;
{ELSE}
  gfbNciCtrl            : ARRAY[1..cMaxNciCh] OF I_Nci_Ctrl;
{END_IF}
END_VAR

// ---- POUs/NCI/I_NciChannel.TcIO
INTERFACE I_NciChannel

(*
===============================================================
Implementation of Tc2_NCI.CfgBuildExt3DGroup

  Builds complete NCI-Group with all configured axes
===============================================================
*)
METHOD BuildGroup : HRESULT
VAR_INPUT
  Execute: BOOL;
END_VAR
END_METHOD

(*
===============================================================
NCI-Group configured axes structure
===============================================================
*)
PROPERTY CfgAxes : Tc2_NCI.NCI_EXT3DGROUP
SET
END_SET
END_PROPERTY

(*
===============================================================
Implementation of Tc2_NCI.CfgReconfigGroup

  remove all axes from NCI-Group
===============================================================
*)
METHOD ClearGroup : HRESULT
VAR_INPUT
  Execute: BOOL;
END_VAR
END_METHOD

METHOD ConfirmHSK : HRESULT
VAR_INPUT
  Execute: BOOL;
END_VAR
END_METHOD

(*
===============================================================
Implementation of Tc2_NCI.ItpDelDtgEx

  DelDTG ( delete distance to go ) wird aus dem NC Programm satzweise aktiviert. 
  Dieses Kommando ermöglicht es, aus der SPS ( TcNci.lib ItpDelDtgEx) den Restweg der aktuellen Geometrie zu löschen. 
  D.h. trifft das Kommando während der Abarbeitung des Satzes ein so wird mit den üblichen Verzögerungsrampen die Bewegung angehalten. 
  Anschließend wird mit dem nächsten Satz im NC Programm fortgefahren.
  Falls das SPS-Kommando nicht während der Ausführung eines Satzes mit angewähltem Restweglöschen eintrifft, wird dieses mit einer Fehlermeldung beantwortet.
  Das Restweglöschen bewirkt immer einen impliziten Dekodierstop, d.h. es erfolgt am Satzende immer ein Genauhalt.
===============================================================
*)
METHOD DelDTG : HRESULT
VAR_INPUT
  Execute: BOOL;
END_VAR
END_METHOD

PROPERTY Error : BOOL
GET
END_GET
END_PROPERTY

METHOD Error_Get : BOOL
END_METHOD

(*
===============================================================
Implementation of Tc2_NCI.ItpEStopEx
===============================================================
*)
METHOD EStop : HRESULT
VAR_INPUT
  Execute: BOOL;
END_VAR
END_METHOD

METHOD GetChannelOverride : real
VAR_INPUT
END_VAR
END_METHOD

METHOD GetItpState : uint
VAR_INPUT
END_VAR
END_METHOD

PROPERTY HSK : BOOL
GET
END_GET
END_PROPERTY

PROPERTY I_AuxAxis : ARRAY[1..GVL_NCI.cAuxAxisCount] OF I_McAxis
SET
END_SET
END_PROPERTY

PROPERTY I_McAxis : array[1..GVL_NCI.cMcAxisCount] of I_McAxis
SET
END_SET
END_PROPERTY

PROPERTY ItpAxes : Tc2_NCI.NCI_EXT3DGROUP
GET
END_GET
END_PROPERTY

(*
===============================================================
Implementation of Tc2_NCI.ItpResetEx2
===============================================================
*)
METHOD ItpReset : HRESULT
VAR_INPUT
  Execute: BOOL;
END_VAR
END_METHOD

METHOD LoadProg : HRESULT
VAR_INPUT
  Execute: BOOL;
END_VAR
END_METHOD

PROPERTY MFunc : INT
GET
END_GET
END_PROPERTY

PROPERTY Override : LREAL
GET
END_GET
SET
END_SET
END_PROPERTY

PROPERTY PathVelo : LREAL
GET
END_GET
END_PROPERTY

PROPERTY pNciChannelRef : POINTER TO ST_NciChannel_Ref
GET
END_GET
END_PROPERTY

PROPERTY Prog : STRING(255)
GET
END_GET
SET
END_SET
END_PROPERTY

(*
===============================================================
Implementation of Tc2_System.ADSREADEX

  reads actual interpreter G-Code Line
===============================================================
*)
METHOD ReadLine : HRESULT
VAR_INPUT
  Execute: BOOL;
END_VAR
//Read G-Code actual Line
VAR_OUTPUT
  ActProgLine: STRING(100);
END_VAR
END_METHOD

(*
===============================================================
Implementation of Tc2_NCI.ItpReadRParamsEx

  read R-Parameter(s) from NCI
===============================================================
*)
METHOD ReadRParams : HRESULT
VAR_INPUT
  Execute :BOOL;
  Addr    :POINTER TO LREAL;  //Adresse der Zielvariablen der zu lesenden Daten. 
        //Dabei werden die Daten direkt ab der angegebenen Adresse von der NC beschrieben  
        //D.h. nIndex ist nicht als Offset zu pAddr zu sehen. Die Daten befinden sich z.B. 
        //in einem Array vom Typ LREAL, das vom Anwender definiert werden muss.
  Index   :DINT;
  Count   :DINT;
END_VAR
END_METHOD

(*
===============================================================
Implementation of Tc2_NCI.ItpStartStopEx

  Start Interpreter
===============================================================
*)
METHOD StartStop : HRESULT
VAR_INPUT
  Start: BOOL;
  Stop: BOOL;
END_VAR
END_METHOD

(*
===============================================================
Implementation of Tc2_NCI.ItpStopOnAfterEStopEx
===============================================================
*)
METHOD StepOnAfterEStop : HRESULT
VAR_INPUT
  Execute: BOOL;
END_VAR
END_METHOD

(*
===============================================================
Implementation of Tc2_NCI.ItpWriteRParamsEx

  write R-Parameter(s) to NCI
===============================================================
*)
METHOD WriteRParams : HRESULT
VAR_INPUT
  Execute :BOOL;
  Addr    :POINTER TO LREAL;  //Adresse der Zielvariablen der Daten. 
        //Dabei werden die Daten direkt ab der angegebenen Adresse von der NC beschrieben  
        //D.h. nIndex ist nicht als Offset zu pAddr zu sehen. Die Daten befinden sich z.B. 
        //in einem Array vom Typ LREAL, das vom Anwender definiert werden muss.
  Index   :DINT;
  Count   :DINT;
END_VAR
END_METHOD

END_INTERFACE

// ---- POUs/NCI/I_Nci_Ctrl.TcIO
INTERFACE I_Nci_Ctrl

PROPERTY ChnId : udint
GET
END_GET
END_PROPERTY

METHOD Cycle
VAR_INPUT
END_VAR
END_METHOD

PROPERTY eCmd : e_Ctrl_NciCommand
GET
END_GET
SET
END_SET
END_PROPERTY

PROPERTY eState : e_Ctrl_NciCommand
GET
END_GET
SET
END_SET
END_PROPERTY

PROPERTY GroupAxisConfig : ST_3D_Group
GET
END_GET
SET
END_SET
END_PROPERTY

PROPERTY I_AuxAxis : array[1..GVL_NCI.cAuxAxisCount] of I_McAxis
GET
END_GET
SET
END_SET
END_PROPERTY

PROPERTY I_McAxis : array[1..GVL_NCI.cMcAxisCount] of I_McAxis
GET
END_GET
SET
END_SET
END_PROPERTY

PROPERTY I_NcChannel : I_NciChannel
GET
END_GET
END_PROPERTY

PROPERTY M_FuncReq : word
GET
END_GET
END_PROPERTY

PROPERTY NcProg : string(255)
GET
END_GET
SET
END_SET
END_PROPERTY

PROPERTY R_Param_Read : ARRAY [0..GVL_NCI.cRParamCount] OF lreal
GET
END_GET
SET
END_SET
END_PROPERTY

PROPERTY R_Param_Write : ARRAY [0..GVL_NCI.cRParamCount] OF lreal
GET
END_GET
SET
END_SET
END_PROPERTY

PROPERTY R_ParamCount : DINT
GET
END_GET
SET
END_SET
END_PROPERTY

PROPERTY R_ParamIndex : DINT
GET
END_GET
SET
END_SET
END_PROPERTY

PROPERTY sCmd : string
GET
END_GET
SET
END_SET
END_PROPERTY

END_INTERFACE

// ---- POUs/NC_AXIS/I_McAxis.TcIO
INTERFACE I_McAxis

PROPERTY pAxisRef : pointer to AXIS_REF
GET
END_GET
END_PROPERTY

PROPERTY Position : LREAL
GET
END_GET
END_PROPERTY

END_INTERFACE

// ---- POUs/MAPPING/MAPPING_in.TcPOU
PROGRAM MAPPING_in
VAR CONSTANT
{IF defined (AXIS_MAP)}
  {info 'MAPPING_in - ACTIVE'}
  bBypassMapping    : BOOL  := FALSE;
{ELSE}
  bBypassMapping    : BOOL  := TRUE;
{END_IF}
END_VAR
VAR
  AxisCTrl              : U_AXIS_CTRL;
  AxisMotionOptions     : U_AXIS_MOTION_OPTIONS;

  AxisGearInData        : U_AXIS_GEAR_IN;
  AxisGearInMultiMaster : U_AXIS_GEAR_IN_MULTIMASTER;
  AxisHoming            : U_AXIS_HOMING;
  AxisParameterWrt      : U_AXIS_NC_PARAMETER;

  nAxis                 : INT;
END_VAR

IF bBypassMapping THEN RETURN; END_IF


FOR nAxis := 1 TO GVL_AXIS_CTRL.gciMaxAxis
DO
  memcpy(ADR(GVL_AXIS_CTRL.gstAxisControl[nAxis].ToPlc),  ADR(AxisCtrl.stCtrl[nAxis]),          SIZEOF(ST_In));
  memcpy(ADR(GVL_AXIS_CTRL.gstMotionOptions[nAxis]),      ADR(AxisMotionOptions.stCtrl[nAxis]), SIZEOF(ST_MotionOptions));
  memcpy(ADR(GVL_AXIS_CTRL.gstAxisGearParam[nAxis]),      ADR(AxisGearInData.stCtrl[nAxis]),    SIZEOF(ST_GearIn));
  memcpy(ADR(GVL_AXIS_CTRL.gstHomeParam[nAxis]),          ADR(AxisHoming.stCtrl[nAxis]),        SIZEOF(ST_HomeParams));

  GVL_AXIS_CTRL.gstAxisParam[nAxis].bRead             := AxisParameterWrt.stState[nAxis].bRead;
  GVL_AXIS_CTRL.gstAxisParam[nAxis].bWrite            := AxisParameterWrt.stState[nAxis].bWrite;
  GVL_AXIS_CTRL.gstAxisParam[nAxis].ParameterNumber   := AxisParameterWrt.stState[nAxis].ParameterNumber;
  GVL_AXIS_CTRL.gstAxisParam[nAxis].rValueWrite       := AxisParameterWrt.stState[nAxis].rValueWrite;
END_FOR

END_PROGRAM

// ---- POUs/MAIN.TcPOU
PROGRAM MAIN
VAR
	uiFrm0_State				AT %I* : UINT;
	uiFrm0_WcState			AT %I* : UINT;
	uiFrm0_InputToggle	AT %I* : UINT;
	uiSlaveCount				AT %I* : UINT;
	uiDevState					AT %I* : UINT;

{IF defined (TEST)}
  {info 'TEST'}
	bSafety_OK					       : BOOL := TRUE;
{ELSE}
	bSafety_OK					AT %I* : BOOL; // Input for TwinSAFE signal for SS1 stop
{END_IF}

	aOut	AT %Q* : BOOL;
	bTic				 : BOOL;
	diCounter		 : DINT;
	imod				 : INT := 10;

	szAxisCtrl, 
	szAxisCtrlPlc, 
	szAxisCtrlC, 
	szNcParam,
	szHomeParam	: UINT;
	iAxisIndex	: INT := 1;
	i						: INT;

	rtrigWriteFile		: R_TRIG;
  tonWriteFile      : TON;
  tWriteFile        : time := t#5s;
END_VAR

// Local time; used for timestamps
GVL_AXIS_CTRL.gfbLocalTime(sLocalTime=> GVL_AXIS_CTRL.gsLocalTime, dtLocalTime=> GVL_AXIS_CTRL.gdtLocalTime);


diCounter := diCounter + 1;

// tic for ADS notification
IF (diCounter MOD imod = 0)
THEN
	bTic          := NOT bTic;
	aOut          := NOT aOut;
END_IF

szAxisCtrl      := SIZEOF(GVL_AXIS_CTRL.gstAxisControl[iAxisIndex]);
szAxisCtrlPlc   := SIZEOF(GVL_AXIS_CTRL.gstAxisControl[iAxisIndex].ToPlc);
szAxisCtrlC     := SIZEOF(GVL_AXIS_CTRL.gstAxisControl[iAxisIndex].FromPlc);
szNcParam       := SIZEOF(GVL_AXIS_CTRL.gstAxisParam[iAxisIndex]);
szHomeParam     := SIZEOF(GVL_AXIS_CTRL.gstHomeParam[iAxisIndex]);

FOR i := 1 TO GVL_AXIS_CTRL.gciMaxAxis
DO
  CASE GVL_AXIS_CTRL.gstAxisControl[i].ToPlc.uiAxisFunctionReq 
  OF
    //-----------------------------------------------------------------------------------------------------------------
    // GearIn
    //-----------------------------------------------------------------------------------------------------------------
    e_AxisFunction.AXIS_GEAR_IN:

      IF(GVL_AXIS_CTRL.gstAxisControl[i].ToPlc.byAxisFuncPara > 0) AND
        (GVL_AXIS_CTRL.gstAxisControl[i].ToPlc.byAxisFuncPara <= GVL_AXIS_CTRL.gciMaxAxis)
      THEN
        // copy index to diag array
        GVL_AXIS_CTRL.gbyAxisIdxGearIn[i]                       := GVL_AXIS_CTRL.gstAxisControl[i].ToPlc.byAxisFuncPara; // FuncParam for GEAR_IN carries array index of master axis
        GVL_AXIS_CTRL.gfbAxisController[i].MasterAxis1          := GVL_AXIS_CTRL.gfbAxisController[GVL_AXIS_CTRL.gbyAxisIdxGearIn[i]].fbAxis.pAxisRef;
        GVL_AXIS_CTRL.gfbAxisController[i].stGear               := GVL_AXIS_CTRL.gstAxisGearParam[i];
        GVL_AXIS_CTRL.gstAxisControl[i].FromPlc.byAxisFuncPara  := GVL_AXIS_CTRL.gbyAxisIdxGearIn[i];
      END_IF


    //-----------------------------------------------------------------------------------------------------------------
    // GearInMultimaster
    //-----------------------------------------------------------------------------------------------------------------
    e_AxisFunction.AXIS_GEAR_IN_MULTIMASTER:

      // Master 1
      IF(GVL_AXIS_CTRL.gstAxisGearMultiMasterParam[i].byAxisIDMaster1 > 0) AND
        (GVL_AXIS_CTRL.gstAxisGearMultiMasterParam[i].byAxisIDMaster1 <= GVL_AXIS_CTRL.gciMaxAxis) 
      THEN
        GVL_AXIS_CTRL.gbyAxisIdxGearInMultiMaster[i,1]          := GVL_AXIS_CTRL.gstAxisGearMultiMasterParam[i].byAxisIDMaster1;
        GVL_AXIS_CTRL.gfbAxisController[i].MasterAxis1          := GVL_AXIS_CTRL.gfbAxisController[GVL_AXIS_CTRL.gstAxisGearMultiMasterParam[i].byAxisIDMaster1].fbAxis.pAxisRef;
      ELSE
        GVL_AXIS_CTRL.gbyAxisIdxGearInMultiMaster[i,1]          := 0;
        GVL_AXIS_CTRL.gfbAxisController[i].MasterAxis1          := 0;
      END_IF

      // Master 2
      IF(GVL_AXIS_CTRL.gstAxisGearMultiMasterParam[i].byAxisIDMaster2 > 0) AND
        (GVL_AXIS_CTRL.gstAxisGearMultiMasterParam[i].byAxisIDMaster2 <= GVL_AXIS_CTRL.gciMaxAxis)	  
      THEN
        GVL_AXIS_CTRL.gbyAxisIdxGearInMultiMaster[i,2]          := GVL_AXIS_CTRL.gstAxisGearMultiMasterParam[i].byAxisIDMaster2;
        GVL_AXIS_CTRL.gfbAxisController[i].MasterAxis2          := GVL_AXIS_CTRL.gfbAxisController[GVL_AXIS_CTRL.gstAxisGearMultiMasterParam[i].byAxisIDMaster2].fbAxis.pAxisRef;
      ELSE
        GVL_AXIS_CTRL.gbyAxisIdxGearInMultiMaster[i,2]          := 0;
        GVL_AXIS_CTRL.gfbAxisController[i].MasterAxis2          := 0;
      END_IF 

      // Master 3
      IF(GVL_AXIS_CTRL.gstAxisGearMultiMasterParam[i].byAxisIDMaster3 > 0) AND
       (GVL_AXIS_CTRL.gstAxisGearMultiMasterParam[i].byAxisIDMaster3 <= GVL_AXIS_CTRL.gciMaxAxis)
      THEN
        GVL_AXIS_CTRL.gbyAxisIdxGearInMultiMaster[i,3]          := GVL_AXIS_CTRL.gstAxisGearMultiMasterParam[i].byAxisIDMaster3;
        GVL_AXIS_CTRL.gfbAxisController[i].MasterAxis3          := GVL_AXIS_CTRL.gfbAxisController[GVL_AXIS_CTRL.gstAxisGearMultiMasterParam[i].byAxisIDMaster3].fbAxis.pAxisRef;
      ELSE
        GVL_AXIS_CTRL.gbyAxisIdxGearInMultiMaster[i,3]          := 0;
        GVL_AXIS_CTRL.gfbAxisController[i].MasterAxis3          := 0;
      END_IF

      // Master 4	 
      IF(GVL_AXIS_CTRL.gstAxisGearMultiMasterParam[i].byAxisIDMaster4 >= 0) AND
        (GVL_AXIS_CTRL.gstAxisGearMultiMasterParam[i].byAxisIDMaster4 <= GVL_AXIS_CTRL.gciMaxAxis)
      THEN
        GVL_AXIS_CTRL.gbyAxisIdxGearInMultiMaster[i,4]          := GVL_AXIS_CTRL.gstAxisGearMultiMasterParam[i].byAxisIDMaster4;
        GVL_AXIS_CTRL.gfbAxisController[i].MasterAxis4          := GVL_AXIS_CTRL.gfbAxisController[GVL_AXIS_CTRL.gstAxisGearMultiMasterParam[i].byAxisIDMaster4].fbAxis.pAxisRef;
      ELSE
        GVL_AXIS_CTRL.gbyAxisIdxGearInMultiMaster[i,4]          := 0;
        GVL_AXIS_CTRL.gfbAxisController[i].MasterAxis4          := 0;
      END_IF

      GVL_AXIS_CTRL.gfbAxisController[i].stGearMultiMaster      := GVL_AXIS_CTRL.gstAxisGearMultiMasterParam[i];


    //-----------------------------------------------------------------------------------------------------------------
    // CamIn
    //-----------------------------------------------------------------------------------------------------------------
    e_AxisFunction.AXIS_CAM_IN:

      IF(GVL_AXIS_CTRL.gstAxisControl[i].ToPlc.byAxisFuncPara > 0) AND
        (GVL_AXIS_CTRL.gstAxisControl[i].ToPlc.byAxisFuncPara <= GVL_AXIS_CTRL.gciMaxAxis)
      THEN
      // copy index to diag array
        GVL_AXIS_CTRL.gbyAxisIdxCamIn[i]                        := GVL_AXIS_CTRL.gstAxisControl[i].ToPlc.byAxisFuncPara; // FuncParam carries array index of master axis
      // assign master axis
        GVL_AXIS_CTRL.gfbAxisController[i].MasterAxis1          := GVL_AXIS_CTRL.gfbAxisController[GVL_AXIS_CTRL.gbyAxisIdxCamIn[i]].fbAxis.pAxisRef;
      // assign CAM parameters
        GVL_AXIS_CTRL.gfbAxisController[i].stCam                := GVL_AXIS_CTRL.gstAxisCamParam[i];
      // copy index to FromPLC structure 
        GVL_AXIS_CTRL.gstAxisControl[i].FromPlc.byAxisFuncPara  := GVL_AXIS_CTRL.gbyAxisIdxCamIn[i];
      END_IF


	
  ELSE  
    GVL_AXIS_CTRL.gbyAxisIdxGearIn[i]                           := 0;

    GVL_AXIS_CTRL.gbyAxisIdxGearInMultiMaster[i,1]              := 0;
    GVL_AXIS_CTRL.gbyAxisIdxGearInMultiMaster[i,2]              := 0;
    GVL_AXIS_CTRL.gbyAxisIdxGearInMultiMaster[i,3]              := 0;
    GVL_AXIS_CTRL.gbyAxisIdxGearInMultiMaster[i,4]              := 0;

    GVL_AXIS_CTRL.gbyAxisIdxCamIn[i]                            := 0;
    GVL_AXIS_CTRL.gfbAxisController[i].MasterAxis1              := 0;
  END_CASE


  //-----------------------------------------------------------------------------------------------------------------
  // Axis cyclic call
  //-----------------------------------------------------------------------------------------------------------------
	GVL_AXIS_CTRL.gfbAxisController[i](	stCtrl	                  := GVL_AXIS_CTRL.gstAxisControl[i].ToPlc,   // global struct to write on 

                                      bSS1						          := bSafety_OK, 
                                      stHomingOptions	          := GVL_AXIS_CTRL.gstHomeParam[i], 
                                      stNcParameter		          := GVL_AXIS_CTRL.gstAxisParam[i],
                                      stMotionOptions           := GVL_AXIS_CTRL.gstMotionOptions[i],

                                      stState					          => GVL_AXIS_CTRL.gstAxisControl[i].FromPlc  // global struct to read from
                                     );   
END_FOR

tonWriteFile(IN := TRUE, PT := tWriteFile);

IF tonWriteFile.Q
THEN
  p_Data.bWriteFile := TRUE;
  tonWriteFile(IN:=FALSE);
END_IF  

//-----------------------------------------------------------------------------------------------------------------
// write message list to file
//-----------------------------------------------------------------------------------------------------------------
p_Data(pList			:= ADR(GVL_AXIS_CTRL.gatMessages),
			 pLocalTime := ADR(GVL_AXIS_CTRL.gdtLocalTime), 
			 bBusy=> );



IF p_Data.bWriteFile AND
   p_Data.bBusy
THEN
  p_Data.bWriteFile := FALSE;
END_IF

P_CopleyWorkAround();

END_PROGRAM

// ---- POUs/MSG/p_Data.TcPOU
PROGRAM p_Data
VAR_INPUT
	bPowerFail		: BOOL;
	bWriteFile		: BOOL;
	bReset				: BOOL;
	pList					: POINTER TO ARRAY[1..GVL_AXIS_CTRL.gciMaxMessage] OF ST_Message;
	pLocalTime		: POINTER TO DT; 
END_VAR
VAR_OUTPUT
	bBusy					: BOOL;
	VisuList		  : ARRAY[1..GVL_AXIS_CTRL.gciMaxMessage] OF ST_Message;
END_VAR
VAR
	diStep 				: DINT;

	rtrigReset		: Tc2_Standard.R_TRIG;
	aWriteList		: ARRAY[1..GVL_AXIS_CTRL.gciMaxMessage] OF ST_Message;
	sWriteData		: STRING(32767);
	sNewLine			: STRING := '$N';
	sTab					: STRING := '$T';
	iCount, 
	iStart, 
	iEnd					: INT;

	fbWrite				: fb_WriteData;
	fbCreateDir		: Tc2_System.FB_CreateDir;
	sTmp          : STRING(256);
	sFilename			: STRING(256);
	sFolderDate		: STRING;
	bFileCreated	: BOOL;

  ivis          : INT;
END_VAR
VAR CONSTANT
	MSG_WRITE_COUNT	: INT := 10;
END_VAR

(* pointer check *)
IF NOT (pList <> 0) OR
	 NOT (pLocalTime <> 0)
THEN
	RETURN;
END_IF

IF (f_FolderDate(pLocalTime) <> sFolderDate)
THEN
	bFileCreated := FALSE;
END_IF


rtrigReset(CLK:= bReset);
IF rtrigReset.Q
THEN
	bReset := FALSE;
	diStep := 0;
END_IF


CASE diStep OF
	0:
		bBusy := FALSE;
    IF bWriteFile
    THEN
      diStep := 5;
		ELSIF (GVL_AXIS_CTRL.giMsgIndex >= MSG_WRITE_COUNT) OR
			     bPowerFail
		THEN
      diStep := 5;
	END_IF
END_CASE
CASE diStep OF
  5:
			memcpy(ADR(aWriteList), pList, SIZEOF(aWriteList));
			memset(pList, 0, SIZEOF(aWriteList));

			bBusy                             := TRUE;
			iStart 	                          := 1;
			iEnd 		                          := SEL((GVL_AXIS_CTRL.giMsgIndex > GVL_AXIS_CTRL.gciMaxMessage),
                                                GVL_AXIS_CTRL.giMsgIndex,
                                                GVL_AXIS_CTRL.gciMaxMessage);

			GVL_AXIS_CTRL.giMsgIndex          := 1;

			fbWrite.bExecute                  := FALSE;

			IF NOT bFileCreated
			THEN
        IF (GVL_AXIS_CTRL.giErrorIndex > 0)
        THEN
          GVL_AXIS_CTRL.giErrorIndex    := 0;
				  diStep                        := 10;
        ELSE
          diStep                        := 250;
        END_IF
			ELSE
        GVL_AXIS_CTRL.giErrorIndex      := 0;
				diStep := 200;
			END_IF
END_CASE
CASE diStep OF
	10:
		fbCreateDir.sPathName := left(GVL_AXIS_CTRL.gcsLogDir,len(GVL_AXIS_CTRL.gcsLogDir)-1);
		fbCreateDir.bExecute  := FALSE;
		diStep := 20;

	20:
		(* create root folder *)
		fbCreateDir.bExecute	:= TRUE;
		IF fbCreateDir.bBusy
		THEN
			diStep := 30;
		END_IF

	30:
		IF NOT fbCreateDir.bBusy
		THEN
			sFolderDate := f_FolderDate(pLocalTime);
			fbCreateDir.sPathName := concat(GVL_AXIS_CTRL.gcsLogDir, sFolderDate);
			fbCreateDir.bExecute  := FALSE;
			diStep := 40;
		END_IF

	40:
		(* create active folder *)
		fbCreateDir.bExecute	:= TRUE;
		IF fbCreateDir.bBusy
		THEN
			diStep := 50;
		END_IF

	50:
		IF NOT fbCreateDir.bBusy
		THEN
			fbCreateDir.bExecute  := FALSE;
			// build complete file path
			sTmp := concat(concat(GVL_AXIS_CTRL.gcsLogFile, sFolderDate),'.txt');
			sTmp := concat('\', sTmp);
			sFilename := concat(fbCreateDir.sPathName, sTmp);
			bFileCreated := TRUE;
			diStep := 200;
		END_IF

END_CASE
CASE diStep OF
	200:
		memset(ADR(sWriteData),0,SIZEOF(sWriteData));
		iCount := iStart;
		diStep := 220;

	220:
		IF aWriteList[iCount].eType > 0
		THEN
      IF (aWriteList[iCount].eType > E_MessageType.eMessageInfo) OR
          GVL_AXIS_CTRL.gbEnableLogging
      THEN
        sTmp := TO_STRING(aWriteList[iCount].eType);
        sTmp := Tc2_Standard.CONCAT(sTmp, sTab);
        sTmp := Tc2_Standard.CONCAT(sTmp, aWriteList[iCount].tTime);
        sTmp := Tc2_Standard.CONCAT(sTmp, sTab);
        sTmp := Tc2_Standard.CONCAT(sTmp, Device_To_String(aWriteList[iCount].eDevice));
        sTmp := Tc2_Standard.CONCAT(sTmp, sTab);
        sTmp := Tc2_Standard.CONCAT(sTmp, TO_STRING(aWriteList[iCount].eSubdevice));
        sTmp := Tc2_Standard.CONCAT(sTmp, sTab);
        sTmp := Tc2_Standard.CONCAT(sTmp, TO_STRING(aWriteList[iCount].iErrorNumber));
        sTmp := Tc2_Standard.CONCAT(sTmp, sTab);
        sTmp := Tc2_Standard.CONCAT(sTmp, aWriteList[iCount].sText);
        sTmp := Tc2_Standard.CONCAT(sTmp, sNewLine);
        f_Builder(ADR(sTmp), ADR(sWriteData), len(sTmp));
      END_IF
		END_IF
		iCount := iCount + 1;
		diStep := 225;

	225:
		IF iCount > iEnd
		THEN
			IF (len(sWriteData) > 0)
			THEN
				diStep := 230;
			ELSE
				diStep := 250;
			END_IF
		ELSE
			diStep := 220;
		END_IF


	230:
		fbWrite.bExecute 	:= TRUE;
		IF fbWrite.bBusy
		THEN
			diStep := 240;
		END_IF

	240:
		IF NOT fbWrite.bBusy
		THEN
			fbWrite.bExecute := FALSE;
			diStep := 250;
		END_IF

	250:
		IF NOT bWriteFile
		THEN
			diStep := 0;
		END_IF
END_CASE

fbWrite(
	bExecute:= , 
	sFileName:= sFilename, 
	psData:= ADR(sWriteData), 
	bBusy=> , 
	bDone=> , 
	bError=> );

fbCreateDir(
	sNetId:= , 
	sPathName:=, 
	ePath:= , 
	bExecute:= , 
	tTimeout:= , 
	bBusy=> , 
	bError=> , 
	nErrId=> );

// copy list for visu
FOR ivis := 1 TO GVL_AXIS_CTRL.giMsgIndex
DO
  VisuList[ivis] := pList^[ivis];
END_FOR

METHOD Device_to_String : string
VAR_INPUT
  eMsgDevice    : e_Device;
END_VAR
VAR
  // first NC Axis, all other Axis are incremented
  nmodAxis            : DINT := 1000;

  // first NCI channel control instance
  nmodNciChannelCtrl  : DINT := 2000;

  // NCI channel
  nmodNciChannel      : DINT := 3000;

  // message function blocks
  nmodData            : DINT := 10000;

  sId                 : STRING := '_ID_';
  nId                 : DINT;
END_VAR

IF (eMsgDevice <= nmodAxis)
THEN
  // general case with no added indices
  Device_to_String := TO_STRING(eMsgDevice);
ELSE

  IF (eMsgDevice > nModData)
  THEN
    nId := eMsgDevice MOD nmodData;
    sId := concat(sId, TO_STRING(nId));
 
    Device_to_String := concat(TO_STRING(e_device.Data), sId);

  ELSIF (eMsgDevice > nmodNciChannel)
  THEN
    nId := eMsgDevice MOD nmodNciChannel;
    sId := concat(sId, TO_STRING(nId));
 
    Device_to_String := concat(TO_STRING(e_device.NciChannel), sId);

  ELSIF (eMsgDevice > nmodNciChannelCtrl)
  THEN
    nId := eMsgDevice MOD nmodNciChannelCtrl;
    sId := concat(sId, TO_STRING(nId));
 
    Device_to_String := concat(TO_STRING(e_device.NciChannelCtrl), sId);

  ELSIF (eMsgDevice > nmodAxis)
  THEN
    nId := eMsgDevice MOD nmodAxis;
    sId := concat(sId, TO_STRING(nId));
 
    Device_to_String := concat(TO_STRING(e_device.Axis), sId);
  ELSE
    Device_to_String := TO_STRING(eMsgDevice);
  END_IF
END_IF
END_METHOD

END_PROGRAM

// ---- POUs/MSG/fb_WriteData.TcPOU
FUNCTION_BLOCK fb_WriteData
VAR_INPUT
	bExecute		: BOOL;
	sFileName		: Tc2_System.T_MaxString; (* filename and ending *)
	psData			: POINTER TO STRING(32767);
END_VAR
VAR_OUTPUT
	bBusy				: BOOL;
	bDone				: BOOL;
	bError			: BOOL;
END_VAR
VAR
	diStep			: DINT;
	udiCounter	: UDINT;

	fbFileOpen		: Tc2_System.FB_FileOpen;
	fbFileWrite		: Tc2_System.FB_FileWrite;
	fbFileClose		: Tc2_System.FB_FileClose;

	sTimeStart		: STRING;
	sTimeEnd			: STRING;
END_VAR

udiCounter := udiCounter + 1;

(* pointer check *)
IF (psData = 0)
THEN
	RETURN;
END_IF

IF NOT bExecute
THEN
	diStep := 0;
END_IF

CASE diStep OF

	0:
		fbFileOpen.bExecute		:= FALSE;
		fbFileWrite.bExecute	:= FALSE;
		fbFileClose.bExecute	:= FALSE;
		bBusy := FALSE;
		bDone := FALSE;
		IF bExecute
		THEN
			sTimeStart := GVL_AXIS_CTRL.gfbLocalTime.sLocalTime;
			bBusy  := TRUE;
			diStep := 10;
		END_IF

	10:
		fbFileOpen.bExecute  := TRUE;
		IF fbFileOpen.bBusy
		THEN
			diStep := 20;
		END_IF

	20:
		IF NOT fbFileOpen.bBusy
		THEN
			fbFileOpen.bExecute  := FALSE;
			fbFileWrite.bExecute := TRUE;
			diStep := 30;
		END_IF

	30:
		IF fbFileWrite.bBusy
		THEN
			diStep := 40;
		END_IF

	40:
		IF NOT fbFileWrite.bBusy
		THEN
			fbFileWrite.bExecute := FALSE;
			fbFileClose.bExecute := TRUE;
			diStep := 50;
		END_IF

	50:
		IF fbFileClose.bBusy
		THEN
			diStep := 60;
		END_IF

	60:
		IF NOT fbFileClose.bBusy
		THEN
			fbFileClose.bExecute := FALSE;
			sTimeEnd 	:= GVL_AXIS_CTRL.gfbLocalTime.sLocalTime;
			diStep 		:= 100;
		END_IF
	
	100:
		bBusy := FALSE;
		bDone := TRUE;
END_CASE


fbFileOpen(
	sNetId:= , 
	sPathName:= sFileName, 
	nMode:= FOPEN_MODEAPPEND, 
	ePath:= PATH_GENERIC, 
	bExecute:= , 
	tTimeout:= T#10S, 
	bBusy=> , 
	bError=> , 
	nErrId=> , 
	hFile=> );

fbFileWrite(
	sNetId:= , 
	hFile:= fbFileOpen.hFile, 
	pWriteBuff:= psData, 
	cbWriteLen:= f_Len(psData), 
	bExecute:= , 
	tTimeout:= T#10S, 
	bBusy=> , 
	bError=> , 
	nErrId=> , 
	cbWrite=> );

fbFileClose(
	sNetId:= , 
	hFile:= fbFileOpen.hFile, 
	bExecute:= , 
	tTimeout:= T#10S, 
	bBusy=> , 
	bError=> , 
	nErrId=> );

bError := fbFileOpen.bError OR fbFileWrite.bError;

END_FUNCTION_BLOCK

// ---- POUs/Functions/f_Len.TcPOU
(*
	string length for len > 255
*)
FUNCTION f_Len : UINT
VAR_INPUT
	pInString		: POINTER TO STRING(32767);
END_VAR
VAR
	Counter			: UINT;
	pInWork			: POINTER TO BYTE;
END_VAR

pInWork := pInString;
Counter := 0;

WHILE (pInWork^ <> 0) AND
			(Counter < 32767)
DO
	Counter := Counter + 1;
	pInWork := pInWork + 1;
END_WHILE

f_Len := Counter;

END_FUNCTION

// ---- POUs/Functions/f_FolderDate.TcPOU
FUNCTION f_FolderDate : STRING
VAR_INPUT
	pLocalTime		: POINTER TO DT;
END_VAR
VAR
	sTmp					: STRING;
END_VAR



IF NOT (pLocalTime <> 0)
THEN
	f_FolderDate := 'NULL';
	RETURN;
END_IF

sTmp := DT_TO_STRING(pLocalTime^);

// cut off #dt literal
sTmp := right(sTmp, len(sTmp)-3);

sTmp := replace(sTmp, '_', 1, 5);
sTmp := replace(sTmp, '_', 1, 8);
//sTmp := replace(sTmp, '_', 1, 11); // hour
//sTmp := replace(sTmp, '_', 1, 14); // minute

sTmp := left(sTmp,10);	// year_month_day
//sTmp := left(sTmp,16); // with hour and minute

f_FolderDate := sTmp;

END_FUNCTION

// ---- POUs/Functions/f_Builder.TcPOU
(*
  string concat for length > 255
*)
FUNCTION f_Builder : Bool
VAR_INPUT
  pInString   : POINTER TO STRING;
  pOutString  : POINTER TO STRING(32767);
  //pOutString  : POINTER TO STRING(16384);
  fLength     : INT;
END_VAR
VAR
  Counter     : DINT;
  pInWork     : POINTER TO BYTE;
  pOutWork    : POINTER TO BYTE;
END_VAR

pOutWork := pOutString;
pInWork := pInString;
Counter := 0;

(*check termination*)
WHILE (pOutWork^ <> 0) AND
      (Counter < 32767)
DO
  Counter := Counter + 1;
  pOutWork := pOutWork + 1;
END_WHILE

(* append only if data fits into output *)
IF (Counter + fLength < 32767)
THEN

  (* append data *)
  FOR Counter := 1 TO fLength
  DO
    pOutWork^ := pInWork^;
    pOutWork := pOutWork + 1;
    pInWork := pInWork + 1;
  END_FOR

  (* terminate *)
  pOutWork := pOutWork + 1;
  pOutWork^ := 0;
END_IF

END_FUNCTION

// ---- POUs/P_CopleyWorkAround.TcPOU
PROGRAM P_CopleyWorkAround
VAR
  bTmp              : BOOL;
  fbTimer           : TON;
  tWait             : TIME := T#6S;
  nIndex, nIdx      : DINT;
  nAxisCount        : DINT := 3;

  aNetId    AT%I*   : AMSNETID;
  nAdr      AT%I*   : ARRAY[1..MAX_AXIS] OF WORD;
  fbEcSetSlaveState : ARRAY[1..MAX_AXIS] OF FB_EcSetSlaveState;

END_VAR
VAR CONSTANT
  MAX_AXIS  : DINT := 10;
END_VAR

nAxisCount := SEL((nAxisCount>MAX_AXIS),nAxisCount,MAX_AXIS);
nAxisCount := SEL((nAxisCount<1),nAxisCount,1);

nIndex := GETCURTASKINDEXEX();
IF _TaskInfo[nIndex].FirstCycle
THEN
  fbTimer.IN := TRUE;
ELSE
  bTmp := TRUE;
  FOR nIdx := 1 TO nAxisCount
  DO
    IF (fbEcSetSlaveState[nIdx].currState.deviceState <> EC_DEVICE_STATE_OP)
    THEN
      bTmp := FALSE;
    END_IF
  END_FOR
  fbTimer.IN := NOT bTmp;
END_IF
fbTimer(PT:= tWait);

FOR nIdx := 1 TO nAxisCount
DO
  fbEcSetSlaveState[nIdx](sNetId:= F_CreateAmsNetId(aNetId), nSlaveAddr:= nAdr[nIdx], bExecute:= fbTimer.Q, reqState:= EC_DEVICE_STATE_OP);
END_FOR

END_PROGRAM

// ---- POUs/NCI.TcPOU
PROGRAM NCI
VAR
  sState          : ARRAY[1..GVL_NCI.cMaxNciCh] OF STRING;


  _idx            : DINT;
  _stAxisIndexItf : ARRAY[1..GVL_NCI.cMaxNciCh] OF ST_Interface_Group;

  _I_McAxis       : ARRAY[1..GVL_NCI.cMaxNciCh]     OF 
                    ARRAY[1..GVL_NCI.cMcAxisCount]  OF I_McAxis;

  _I_AuxAxis      : ARRAY[1..GVL_NCI.cMaxNciCh]     OF 
                    ARRAY[1..GVL_NCI.cAuxAxisCount] OF I_McAxis;
END_VAR


IF NOT GVL_NCI.cNci
THEN
  FOR _idx := 1 TO GVL_NCI.cMaxNciCh
  DO
    GVL_NCI.gstChannelState[_idx].eState        := e_Ctrl_NciCommand.NO_NCI;
  END_FOR
  RETURN;

ELSE
  FOR _idx := 1 TO GVL_NCI.cMaxNciCh
  DO
    IF NOT (GVL_NCI.gstAxisConfig[_idx].nXAxisId > 0) OR
       NOT (GVL_NCI.gstAxisConfig[_idx].nYAxisId > 0) OR
       NOT (GVL_NCI.gstAxisConfig[_idx].nZAxisId > 0)
    THEN
      GVL_NCI.gstChannelState[_idx].eState      := e_Ctrl_NciCommand.NO_AXIS_GROUP; // no valid NC AxisId
      sState[_idx]                              := TO_STRING(_idx);
      sState[_idx]                              := concat(sState[_idx], ': no valid NC AxisId');
      RETURN;
    END_IF
  END_FOR

  FOR _idx := 1 TO GVL_NCI.cMaxNciCh
  DO
    IF NOT (GVL_NCI.gstAxisIndex[_idx].nXAxisIdx > 0) OR
       NOT (GVL_NCI.gstAxisIndex[_idx].nYAxisIdx > 0) OR
       NOT (GVL_NCI.gstAxisIndex[_idx].nZAxisIdx > 0) OR
           (GVL_NCI.gstAxisIndex[_idx].nXAxisIdx > TO_UDINT(GVL_AXIS_CTRL.gciMaxAxis)) OR
           (GVL_NCI.gstAxisIndex[_idx].nYAxisIdx > TO_UDINT(GVL_AXIS_CTRL.gciMaxAxis)) OR
           (GVL_NCI.gstAxisIndex[_idx].nZAxisIdx > TO_UDINT(GVL_AXIS_CTRL.gciMaxAxis))
    THEN
      GVL_NCI.gstChannelState[_idx].eState      := e_Ctrl_NciCommand.NO_AXIS_INDEX; // no valid fb_AxisController[] index
      sState[_idx]                              := TO_STRING(_idx);
      sState[_idx]                              := concat(sState[_idx], ': no valid fb_AxisController[] index');
      RETURN;
    END_IF
  END_FOR
END_IF

FOR _idx := 1 TO GVL_NCI.cMaxNciCh
DO
  // NCI axis configuration --> NC AxisId used
  GVL_NCI.gfbNciCtrl[_idx].GroupAxisConfig      := GVL_NCI.gstAxisConfig[_idx];


  // fb_AxisController.fbAxis I_McAxis configuration --> index of gfbAxisController is used
  IF (GVL_NCI.gstAxisIndex[_idx].nXAxisIdx > 0)
  THEN
    _stAxisIndexItf[_idx].I_Idx_XAxis           := GVL_AXIS_CTRL.gfbAxisController[GVL_NCI.gstAxisIndex[_idx].nXAxisIdx].fbAxis;
  END_IF

  IF (GVL_NCI.gstAxisIndex[_idx].nYAxisIdx > 0)
  THEN
    _stAxisIndexItf[_idx].I_Idx_YAxis           := GVL_AXIS_CTRL.gfbAxisController[GVL_NCI.gstAxisIndex[_idx].nYAxisIdx].fbAxis;
  END_IF

  IF (GVL_NCI.gstAxisIndex[_idx].nZAxisIdx > 0)
  THEN
    _stAxisIndexItf[_idx].I_Idx_ZAxis           := GVL_AXIS_CTRL.gfbAxisController[GVL_NCI.gstAxisIndex[_idx].nZAxisIdx].fbAxis;
  END_IF

  IF (GVL_NCI.gstAxisIndex[_idx].nQ1AxisIdx > 0)
  THEN
    _stAxisIndexItf[_idx].I_Idx_Q1Axis          := GVL_AXIS_CTRL.gfbAxisController[GVL_NCI.gstAxisIndex[_idx].nQ1AxisIdx].fbAxis;
  END_IF

  IF (GVL_NCI.gstAxisIndex[_idx].nQ2AxisIdx > 0)
  THEN
    _stAxisIndexItf[_idx].I_Idx_Q2Axis          := GVL_AXIS_CTRL.gfbAxisController[GVL_NCI.gstAxisIndex[_idx].nQ2AxisIdx].fbAxis;
  END_IF

  IF (GVL_NCI.gstAxisIndex[_idx].nQ3AxisIdx > 0)
  THEN
    _stAxisIndexItf[_idx].I_Idx_Q3Axis          := GVL_AXIS_CTRL.gfbAxisController[GVL_NCI.gstAxisIndex[_idx].nQ3AxisIdx].fbAxis;
  END_IF

  IF (GVL_NCI.gstAxisIndex[_idx].nQ4AxisIdx > 0)
  THEN
    _stAxisIndexItf[_idx].I_Idx_Q4Axis          := GVL_AXIS_CTRL.gfbAxisController[GVL_NCI.gstAxisIndex[_idx].nQ4AxisIdx].fbAxis;
  END_IF

  IF (GVL_NCI.gstAxisIndex[_idx].nQ5AxisIdx > 0)
  THEN
    _stAxisIndexItf[_idx].I_Idx_Q5Axis          := GVL_AXIS_CTRL.gfbAxisController[GVL_NCI.gstAxisIndex[_idx].nQ5AxisIdx].fbAxis;
  END_IF


  _I_McAxis[_idx][1]                            := _stAxisIndexItf[_idx].I_Idx_XAxis;
  _I_McAxis[_idx][2]                            := _stAxisIndexItf[_idx].I_Idx_YAxis;
  _I_McAxis[_idx][3]                            := _stAxisIndexItf[_idx].I_Idx_ZAxis;

  _I_AuxAxis[_idx][1]                           := _stAxisIndexItf[_idx].I_Idx_Q1Axis;
  _I_AuxAxis[_idx][2]                           := _stAxisIndexItf[_idx].I_Idx_Q2Axis;
  _I_AuxAxis[_idx][3]                           := _stAxisIndexItf[_idx].I_Idx_Q3Axis;
  _I_AuxAxis[_idx][4]                           := _stAxisIndexItf[_idx].I_Idx_Q4Axis;
  _I_AuxAxis[_idx][5]                           := _stAxisIndexItf[_idx].I_Idx_Q5Axis;

  GVL_NCI.gfbNciCtrl[_idx].I_McAxis             := _I_McAxis[_idx];
  GVL_NCI.gfbNciCtrl[_idx].I_AuxAxis            := _I_AuxAxis[_idx];

  // R Parameter properties
  GVL_NCI.gfbNciCtrl[_idx].R_ParamIndex         := GVL_NCI.gstRParameter[_idx]._nStart;
  GVL_NCI.gfbNciCtrl[_idx].R_ParamCount         := GVL_NCI.gstRParameter[_idx]._nCount;
  GVL_NCI.gfbNciCtrl[_idx].R_Param_Read         := GVL_NCI.gstRParameter[_idx]._rRParamsRead;
  GVL_NCI.gfbNciCtrl[_idx].R_Param_Write        := GVL_NCI.gstRParameter[_idx]._rRParamsWrite;

  // ProgName for channel
  GVL_NCI.gfbNciCtrl[_idx].NcProg               := GVL_NCI.gsProgName[_idx];

  // check REAL value to avoid exception
  IF NOT IsFinite(F_Real(GVL_NCI.gstChannelCtrl[_idx].rOverride))
  THEN
    GVL_NCI.gfbNciCtrl[_idx].I_NcChannel.Override := 0.0;
  ELSE
    GVL_NCI.gfbNciCtrl[_idx].I_NcChannel.Override := GVL_NCI.gstChannelCtrl[_idx].rOverride;
  END_IF



  // call nci channel controller
  GVL_NCI.gfbNciCtrl[_idx].eCmd                 := GVL_NCI.gstChannelCtrl[_idx].eCmd;
  GVL_NCI.gfbNciCtrl[_idx].Cycle();




  // write states onto global struct
  GVL_NCI.gstChannelState[_idx].eState          := GVL_NCI.gfbNciCtrl[_idx].eState;
  GVL_NCI.gstChannelState[_idx].nItpState       := GVL_NCI.gfbNciCtrl[_idx].I_NcChannel.GetItpState();
  GVL_NCI.gstChannelState[_idx].rAxisOverride   := GVL_NCI.gfbNciCtrl[_idx].I_NcChannel.GetChannelOverride();
  GVL_NCI.gstChannelState[_idx].bMFuncReq       := GVL_NCI.gfbNciCtrl[_idx].I_NcChannel.HSK;
  GVL_NCI.gstChannelState[_idx].nMFunc          := TO_WORD(GVL_NCI.gfbNciCtrl[_idx].I_NcChannel.MFunc);


  GVL_NCI.gsProgNameActive[_idx]                := GVL_NCI.gfbNciCtrl[_idx].I_NcChannel.Prog;
  sState[_idx]                                  := GVL_NCI.gfbNciCtrl[_idx].sCmd;
END_FOR

END_PROGRAM

// ---- POUs/_FunctionBlocks/FB_AxisController.TcPOU
FUNCTION_BLOCK FB_AxisController
VAR_INPUT
	stCtrl					      : ST_In;
	bSS1						      : BOOL := TRUE; // can be used by Safety Alias device
END_VAR
VAR_OUTPUT
	stState					      : ST_Out;
	bXenaxDrive			      : BOOL;
	bSercosAxis			      : BOOL;	// SERCOS encodertype
END_VAR
VAR_IN_OUT
	stHomingOptions	      : ST_HomeParams;
	stNcParameter		      : ST_NcParam;
  stMotionOptions       : ST_MotionOptions;
END_VAR
VAR
	bInit								  : BOOL;
	uiState,
	uiInitState,
	iSizeOut,
	iSizeIn,
  uiStateSS1  				  : UINT;
	sAxisName						  : STRING;
	eState							  : e_AxisFunction;
	eStateOld						  : e_AxisFunction;
	eStateActive				  : e_AxisFunction;
	eStateExec					  : e_AxisFunction; // for logging execution state only
	eStateExecOld				  : e_AxisFunction; // for logging execution state only

  sState, 
  sStateOld, 
  sStateExec            : STRING(256);

	fbAxis							  : FB_McPtpAxis;
	fbResetSercos				  : fb_ResetSercos;					// SOE Reset for Sercos Axis (e.g. AX5000)
	fbXenaxHoming				  : FB_XenaxEtherCATHoming; // for Jenny Science, the homing has to be switched to Xenax
	fbCoeRead						  : Tc2_MC2_Drive.FB_CoERead;

  fbGearIn              : Tc2_MC2.MC_GearIn;
  fbGearInMultiMaster   : Tc2_MC2.MC_GearInMultiMaster;
  fbGearOut             : Tc2_MC2.MC_GearOut;
  _pAxis1               : POINTER TO Tc2_MC2.AXIS_REF;
  _pAxis2               : POINTER TO Tc2_MC2.AXIS_REF;
  _pAxis3               : POINTER TO Tc2_MC2.AXIS_REF;
  _pAxis4               : POINTER TO Tc2_MC2.AXIS_REF;
  _stGearIn             : st_GearIn;
  _stGearInMultiMaster  : st_GearInMultiMaster;	  

{IF defined (CAM)}
  {info 'CAMMING active'}
  _bCamming             : BOOL := TRUE;
  fbCamIn               : Tc2_MC2_Camming.MC_CamIn;
  fbCamOut              : Tc2_MC2_Camming.MC_CamOut;
{ELSE}
  {info 'CAMMING NOT active'}
  _bCamming             : BOOL := FALSE;
  fbCamIn               : FB_CamIn_empty;
  fbCamOut              : FB_CamOut_Empty;
{END_IF}

	_stCamIn              : st_CamIn;

	sDriveType					  : STRING(256); // manufacturer device name CoE 16#1008

	bHomeSensor					  AT %I* : BOOL;
	bLimitMin					    AT %I* : BOOL;
	bLimitMax					    AT %I* : BOOL;

	bFastStop						  AT %Q* : BOOL;
{attribute 'displaymode':='bin'}
	udiDriveInput				  AT %I* : UDINT;
	bDriveInputCal			  : BOOL;
	stMcOut							  : Tc2_MC2.ST_McOutputs;

	tUpdate			          : TIME := T#10S;
  tonTimeout            : Tc2_Standard.TON;
	tonWait			          : Tc2_Standard.TON;
	tonWaitSeq	          : Tc2_Standard.TON;

	_stStatusCompact	    : ST_AxisStatusCompact;
	bHasLagMonitoring	    : BOOL;

	rSetPos, 
  rTmp 		              : LREAL;

	stMsg				          : ST_Message;
 {attribute 'hide'} 
	st_AxisREF_Dummy	    : Tc2_MC2.AXIS_REF;
 {attribute 'hide'}
  mcResetMaster         : Tc2_MC2.MC_Reset;

  eBufferState          : e_AxisFunction;
END_VAR
VAR CONSTANT
	sXenax			: STRING := 'XENAX Xvi';
END_VAR

(*
-------------------------------------------------------------------------------
	update AxisRef and assign CalibrationCam
-------------------------------------------------------------------------------
*)
fbAxis();
fbAxis.SpeedOverride := stCtrl.rOverride;

IF NOT bInit
THEN
  Axis_Init();
END_IF

(*
-------------------------------------------------------------------------------
	NaN INF check
-------------------------------------------------------------------------------
*)
IF NOT IsFinite(F_LReal(stCtrl.rSetPos))
THEN
	stCtrl.rSetPos := 0.0;
END_IF

IF NOT IsFinite(F_LReal(stCtrl.rSetVelo))
THEN
	stCtrl.rSetVelo := 0.0;
END_IF

IF NOT IsFinite(F_LReal(stCtrl.rAcc))
THEN
	stCtrl.rAcc := 0.0;
END_IF

IF NOT IsFinite(F_LReal(stCtrl.rDec))
THEN
	stCtrl.rDec := 0.0;
END_IF

IF NOT IsFinite(F_LReal(stCtrl.rOverride))
THEN
	stCtrl.rOverride := 0.0;
END_IF



(*
-------------------------------------------------------------------------------
	assign CalibrationCam
-------------------------------------------------------------------------------
*)

IF stHomingOptions.SimulateHomeSensor THEN
	IF fbAxis.pAxisRef^.NcToPlc.HomingState < 4 THEN
		bDriveInputCal := TRUE;
	ELSE
		bDriveInputCal := FALSE;
	END_IF
ELSIF stHomingOptions.HomeOnLimitMin THEN
	bDriveInputCal := bLimitMin XOR stHomingOptions.InvertHomeSensor;
ELSIF stHomingOptions.HomeOnLimitMax THEN
	bDriveInputCal := bLimitMax XOR stHomingOptions.InvertHomeSensor;
ELSE
	bDriveInputCal := bHomeSensor XOR stHomingOptions.InvertHomeSensor;
END_IF

fbAxis.CalibrationCam := ADR(bDriveInputCal);

(*
-------------------------------------------------------------------------------
	assign Enable Feed Fw and Feed Bw
-------------------------------------------------------------------------------
*)

IF NOT(stHomingOptions.UseLimitMin) THEN
	fbAxis.FeedEnable_Negative := TRUE;
ELSIF stHomingOptions.HomeOnLimitMin AND fbAxis.pAxisRef^.NcToPlc.HomingState > 0 THEN	
	fbAxis.FeedEnable_Negative := TRUE;
ELSE	
	fbAxis.FeedEnable_Negative := NOT(bLimitMin XOR stHomingOptions.InvertLimitMin);
END_IF

IF NOT(stHomingOptions.UseLimitMax) THEN
	fbAxis.FeedEnable_Positive := TRUE;
ELSIF stHomingOptions.HomeOnLimitMax AND fbAxis.pAxisRef^.NcToPlc.HomingState > 0 THEN	
	fbAxis.FeedEnable_Positive := TRUE;
ELSE	
	fbAxis.FeedEnable_Positive := NOT(bLimitMax XOR stHomingOptions.InvertLimitMax);
END_IF

bFastStop                   := stCtrl.bFastStop;

IF NOT bInit
THEN
	RETURN;
END_IF

(*
-------------------------------------------------------------------------------
	get axis function from interface
-------------------------------------------------------------------------------
*)
stState.bError	            := fbAxis.pAxisRef^.Status.Error; // forward error bit from Axis

eState := stCtrl.uiAxisFunctionReq;

IF (eState <> eStateOld) OR
   (eState = 0)
THEN
  fbAxis.Clear();
  stState.byAxisFuncPara    := 0; // clear mirrored value from ctrl

  stState.bReady            := FALSE;
  stState.bBusy             := FALSE;
  stState.bError            := FALSE;

  eStateExec	              := eState; // clear execution state for logging
  stState.uiErrorId	        := 0;
  stMsg.sText               := '';

  uiState := uiStateSS1     := 0; // reset SS1 state when safety input is back
END_IF


(*
-------------------------------------------------------------------------------
	- get axis SS1 stop
  - else, regular use of axis
-------------------------------------------------------------------------------
*)
IF NOT bSS1
THEN
  // SS1 stop use only
  Axis_Stop_SS1();

  CASE eState OF

    e_AxisFunction.AXIS_DISABLE:
      Axis_Disable();

    e_AxisFunction.AXIS_RESET:
      Axis_Reset_SS1();

    e_AxisFunction.AXIS_PARAMETER:
      Axis_Parameter();

    e_AxisFunction.AXIS_GEAR_OUT:
      Axis_Gear_Out();

    e_AxisFunction.AXIS_CAM_OUT:
      Axis_Cam_Out();

  END_CASE

ELSE

  // regular use
  CASE eState OF
  
    e_AxisFunction.AXIS_DISABLE:
      Axis_Disable();
  
    e_AxisFunction.AXIS_IDLE:
      stState.bReady := NOT fbAxis.pAxisRef^.Status.Error AND 
                        fbAxis.pAxisRef^.Status.ControlLoopClosed;
      Axis_Idle();
  
    e_AxisFunction.AXIS_ENABLE:
      Axis_Enable();  
  
    e_AxisFunction.AXIS_HOME:
      Axis_Home();
  
    e_AxisFunction.AXIS_MOVE_POS:
      Axis_Move_Pos();
  
    e_AxisFunction.AXIS_MOVE_VELO:
      Axis_Move_Velo();
  
    e_AxisFunction.AXIS_RESET:
      Axis_Reset();
  
    e_AxisFunction.AXIS_HALT:
      Axis_Halt();
  
    e_AxisFunction.AXIS_STOP:
      Axis_Stop();
  
    e_AxisFunction.AXIS_MOVE_BUFFER:
      Axis_Move_Buffer();

    e_AxisFunction.AXIS_MOVE_BUFFER_VELO:
      Axis_Move_Buffer_Velocity();
  
    e_AxisFunction.AXIS_PARAMETER:
      Axis_Parameter();
  
    e_AxisFunction.AXIS_GEAR_IN:
      Axis_Gear_In();
  
    e_AxisFunction.AXIS_GEAR_OUT:
      Axis_Gear_Out();
  
    e_AxisFunction.AXIS_GEAR_IN_MULTIMASTER:
      Axis_Gear_In_Multimaster();
  
    e_AxisFunction.AXIS_CAM_IN:
      Axis_Cam_In();
      
  
    e_AxisFunction.AXIS_CAM_OUT:
      Axis_Cam_Out();
  
  ELSE
    // axis function is not available
    stState.bReady          := FALSE;
    stState.bBusy           := FALSE;
    eStateActive 	          := eState + e_AxisFunction.ERROR;
    eStateExec		          := e_AxisFunction.ERROR;
    stState.bError          := TRUE;
    stState.uiErrorId       := 9999;
  END_CASE
  
  (*
  -------------------------------------------------------------------------------
    Xenax drive homing
  -------------------------------------------------------------------------------
  *)
  IF bXenaxDrive
  THEN
    fbXenaxHoming(
      bExecute:= , 
      bAbort:= , 
      Axis:= fbAxis.pAxisRef^, 
      Done=> , 
      Busy=> , 
      Error=> , 
      ErrorId=> );
  END_IF
END_IF // bSS1 = true


(*
-------------------------------------------------------------------------------
	Output Data
-------------------------------------------------------------------------------
*)
// Check CopntrolLoop
IF fbAxis.pAxisRef^.Status.ControlLoopClosed
THEN
  stState.bEnabled          := TRUE;
ELSE
  stState.bEnabled          := FALSE;
END_IF

stState.bStandstill         := fbAxis.pAxisRef^.Status.NotMoving;

// HAUD
// 2023_05_26
// REAL datatype change to LREAL
stState.rActPos             := (fbAxis.pAxisRef^.NcToPlc.ActPos);
stState.rActVelo            := (fbAxis.pAxisRef^.NcToPlc.ActVelo);
stState.rPosDiff            := (fbAxis.pAxisRef^.NcToPlc.PosDiff);

IF (stState.rActPos < stCtrl.rSetPos + fbAxis.stTargetPositionWindow.fValue) AND
   (stState.rActPos > stCtrl.rSetPos - fbAxis.stTargetPositionWindow.fValue) AND
    stState.bStandstill
THEN
  stState.bInTarget         := TRUE;
ELSE
  stState.bInTarget         := FALSE;
END_IF

stState.uiAxisFunctionState := eStateActive;

// HAUD
// 2023 04 05
// copy CoupleState from axis
stState.dwCoupleState       := fbAxis.pAxisRef^.NcToPlc.CoupleState;

sState                      := TO_STRING(eState);
sStateExec                  := TO_STRING(eStateExec);

IF (eStateOld <> eState) AND bInit
THEN
  sStateOld                 := TO_STRING(eStateOld);
  stMsg.eType               := E_MessageType.eMessageInfo;
  stMsg.eDevice             := E_Device.Axis + TO_DINT(fbAxis.pAxisRef^.NcToPlc.AxisId);
  stMsg.eSubdevice          := e_Subdevice.AxisMode;
  stMsg.iErrorNumber        := fbAxis.pAxisRef^.NcToPlc.AxisId;
  stMsg.sText               := 'change ';
  stMsg.sText               := Tc2_Standard.CONCAT(stMsg.sText, sStateOld);
  stMsg.sText               := Tc2_Standard.CONCAT(stMsg.sText, ' to ');
  stMsg.sText               := Tc2_Standard.CONCAT(stMsg.sText, sState);
  f_MessageSet(stMsg);
END_IF

IF (eStateExecOld <> eStateExec) AND bInit
THEN
  stMsg.eType               := E_MessageType.eMessageInfo;
  stMsg.eDevice             := E_Device.Axis + TO_DINT(fbAxis.pAxisRef^.NcToPlc.AxisId);
  stMsg.eSubdevice          := e_Subdevice.AxisMode;
  stMsg.iErrorNumber        := fbAxis.pAxisRef^.NcToPlc.AxisId;
  stMsg.sText               := Tc2_Standard.CONCAT(sState, ' function: ');
  stMsg.sText               := Tc2_Standard.CONCAT(stMsg.sText, TO_STRING(eStateExec));
  f_MessageSet(stMsg);
END_IF

eStateOld                   := eState;
eStateExecOld               := eStateExec;

ACTION Axis_Cam_In:
CASE uiState OF
  0:
    eStateActive            := eState;
    stState.bBusy           := TRUE;
    stState.bReady          := FALSE;

    IF (_pAxis1 <> 0)
    THEN
      fbCamIn(Master        := _pAxis1^, 
              Slave         := fbAxis.pAxisRef^, 
              Execute       := FALSE);
 
      uiState               := 1;

    ELSE
      stMsg.eType           := E_MessageType.eMessageError;
      stMsg.eDevice         := e_Device.Axis + TO_DINT(fbAxis.pAxisRef^.NcToPlc.AxisId);
      stMsg.eSubdevice      := e_Subdevice.fbCamIn;
      stMsg.iErrorNumber    := 666;
      stMsg.sText           := 'Pointer to Masteraxis null';

      f_MessageSet(stMsg);
      stState.uiErrorId		  := TO_UDINT(stMsg.iErrorNumber);

      uiState               :=99;
    END_IF
END_CASE
CASE uiState OF
  1:
  IF NOT (_pAxis1^.Status.Error)
	THEN
		uiState				:= 10;
	ELSE
		mcResetMaster(
					Axis:= _pAxis1^, 
					Execute:= FALSE);
		uiState				:= 2;
	END_IF
END_CASE
CASE uiState OF
  2:
		mcResetMaster(
				Axis:= _pAxis1^, 
				Execute:= TRUE);
	IF mcResetMaster.Done
	THEN
		uiState				:= 0;
	END_IF
END_CASE
CASE uiState OF
  10:
    eStateActive            := eState + e_AxisFunction.AXIS_BUSY;
    eStateExec	            := e_AxisFunction.AXIS_BUSY;

    fbCamIn(Master          := _pAxis1^, 
            Slave           := fbAxis.pAxisRef^, 
            Execute         := TRUE,
            MasterOffset    := _stCamIn.MasterOffset,
            SlaveOffset     := _stCamIn.SlaveOffset,
            MasterScaling   := _stCamIn.MasterScaling,
            SlaveScaling    := _stCamIn.SlaveScaling,
            StartMode       := _stCamIn.StartMode,
            CamTableID      :=_StCamIn.CamTableID);

    IF NOT fbCamIn.Error
    THEN
      IF fbCamIn.InSync
      THEN
        fbCamIn(Master      := _pAxis1^, 
                Slave       := fbAxis._AxisRef, 
                Execute     := FALSE);

        uiState             := 20;
      END_IF
    ELSE
      stMsg.eType           := E_MessageType.eMessageError;
      stMsg.eDevice         := e_Device.Axis + TO_DINT(fbAxis.pAxisRef^.NcToPlc.AxisId);
      stMsg.eSubdevice      := e_Subdevice.fbCamIn;
      stMsg.iErrorNumber    := fbCamIn.ErrorID;
      stMsg.sText           := SEL((_bCamming), 'function not activated with Compiler def CAM', 'error while cam in');

      f_MessageSet(stMsg);

      stState.uiErrorId		  := fbCamIn.ErrorID;

      fbCamIn(Master        := _pAxis1^, 
              Slave         := fbAxis.pAxisRef^, 
              Execute       := FALSE);

      uiState               := 99;
    END_IF
END_CASE
CASE uiState OF
  20:
    stState.bBusy           := FALSE;
    eStateActive            := eState + e_AxisFunction.AXIS_DONE;
    eStateExec	            := e_AxisFunction.AXIS_DONE;

  99:
    stState.bError          := TRUE;
    stState.bBusy           := FALSE;
    eStateActive            := eState + e_AxisFunction.ERROR;
    eStateExec	            := e_AxisFunction.ERROR;
END_CASE
END_ACTION

ACTION Axis_Cam_Out:
CASE uiState OF
  0:
    eStateActive            := eState;
    stState.bBusy           := TRUE;
    stState.bReady          := FALSE;

    fbCamOut(Slave          := fbAxis.pAxisRef^, 
             Execute        := FALSE);

    stMsg.eType 				    := E_MessageType.eMessageInfo;
    stMsg.eDevice 			    := E_Device.Axis  + TO_DINT(fbAxis.pAxisRef^.NcToPlc.AxisId);;
    stMsg.eSubdevice 		    := e_Subdevice.fbCamOut;
    stMsg.iErrorNumber 	    := fbAxis.pAxisRef^.NcToPlc.AxisId;
    stMsg.sText					    := concat('Start CamOut ',TO_STRING(fbAxis.pAxisRef^.NcToPlc.CoupleState));
    f_MessageSet(stMsg);

    // HAUD 2023 04 05
    IF fbAxis.pAxisRef^.Status.Coupled
    THEN
      uiState               := 10;
    ELSE
      uiState               := 20;
      stMsg.eType 				  := E_MessageType.eMessageInfo;
      stMsg.eDevice 			  := E_Device.Axis + TO_DINT(fbAxis.pAxisRef^.NcToPlc.AxisId);;
      stMsg.eSubdevice 		  := e_Subdevice.fbCamOut;
      stMsg.iErrorNumber 	  := 0;
      stMsg.sText           := 'Axis not coupled, ignore function ';
      f_MessageSet(stMsg);
    END_IF
END_CASE
CASE uiState OF
  10:
    eStateActive            := eState + e_AxisFunction.AXIS_BUSY;
    eStateExec	            := e_AxisFunction.AXIS_BUSY;

    fbCamOut(Slave          := fbAxis.pAxisRef^, 
             Execute        := TRUE);

    IF fbCamOut.Error
    THEN
      // HAUD 2023 03 31
      IF NOT fbAxis.pAxisRef^.Status.Coupled
      THEN
        uiState             := 20;
        stMsg.eType 				:= E_MessageType.eMessageWarn;
        stMsg.eDevice 			:= E_Device.Axis + TO_DINT(fbAxis.pAxisRef^.NcToPlc.AxisId);;
        stMsg.eSubdevice 		:= e_Subdevice.fbCamOut;
        stMsg.iErrorNumber 	:= fbCamOut.ErrorID;
        stMsg.sText         := 'Axis not coupled, ignore fb_CamOut error ';
        f_MessageSet(stMsg);

        fbCamOut(Slave      := fbAxis.pAxisRef^, 
                 Execute    := FALSE);
      ELSE
        uiState             := 0;
        // ignore error if axis is coupled; retry      
        stMsg.eType 				:= E_MessageType.eMessageWarn;
        stMsg.eDevice 			:= E_Device.Axis + TO_DINT(fbAxis.pAxisRef^.NcToPlc.AxisId);;
        stMsg.eSubdevice 		:= e_Subdevice.fbCamOut;
        stMsg.iErrorNumber 	:= fbCamOut.ErrorID;
        stMsg.sText         := 'Axis coupled, retry ';
        f_MessageSet(stMsg);
      END_IF
    ELSIF fbCamOut.Done
    THEN
      stMsg.eType 				  := E_MessageType.eMessageInfo;
      stMsg.eDevice 			  := E_Device.Axis + TO_DINT(fbAxis.pAxisRef^.NcToPlc.AxisId);;
      stMsg.eSubdevice 		  := e_Subdevice.fbCamOut;
      stMsg.iErrorNumber 	  := 0;
      stMsg.sText					  := 'fbCamOutDone ';

      f_MessageSet(stMsg);

      uiState               := 20;

      fbCamOut(Slave        := fbAxis.pAxisRef^, 
               Execute      := FALSE);

    ELSIF NOT fbAxis.pAxisRef^.Status.Coupled
    THEN
      stMsg.eType 				  := E_MessageType.eMessageInfo;
      stMsg.eDevice 			  := E_Device.Axis + TO_DINT(fbAxis.pAxisRef^.NcToPlc.AxisId);;
      stMsg.eSubdevice 		  := e_Subdevice.fbCamOut;
      stMsg.iErrorNumber 	  := 0;
      stMsg.sText					  := 'AxisRef not coupled ';

      f_MessageSet(stMsg);

      uiState               := 20;

      fbCamOut(Slave        := fbAxis.pAxisRef^, 
               Execute      := FALSE);
    END_IF
END_CASE
CASE uiState OF
  20:
    stState.bBusy           := FALSE;
    eStateActive            := eState + e_AxisFunction.AXIS_DONE;
    eStateExec	            := e_AxisFunction.AXIS_DONE;

  99:
    stState.bError          := TRUE;
    stState.bBusy           := FALSE;
    eStateActive            := eState + e_AxisFunction.ERROR;
    eStateExec	            := e_AxisFunction.ERROR;
END_CASE
END_ACTION

ACTION Axis_Disable:


eStateActive            := eState;
eStateExec	            := e_AxisFunction.AXIS_BUSY;

tonTimeout(IN           :=FALSE, 
           PT           := tUpdate);

fbAxis.Enable 		      := FALSE;
stState.bTimeout 	      := FALSE;

IF NOT fbAxis.pAxisRef^.Status.ControlLoopClosed
THEN
  eStateActive          := eState + e_AxisFunction.AXIS_DONE;
  eStateExec	          := e_AxisFunction.AXIS_DONE;
END_IF
END_ACTION

ACTION Axis_Enable:

stState.bBusy               := TRUE;
eStateActive                := eState + e_AxisFunction.AXIS_BUSY;
eStateExec	                := e_AxisFunction.AXIS_BUSY;

tonTimeout(IN               := TRUE, 
           PT               := tUpdate);

fbAxis.Enable               := TRUE;

// check if Axis is active
IF fbAxis.pAxisRef^.Status.ControlLoopClosed
THEN
  stState.bTimeout          := FALSE;

  tonTimeout(IN             := FALSE);

  uiState                   := 20;

ELSIF tonTimeout.Q
THEN
  stState.bTimeout          := TRUE;
  stState.uiErrorId         := fbAxis.pAxisRef^.NcToPlc.ErrorCode;

  tonTimeout(IN             := FALSE);

  fbAxis.Enable             := FALSE;

  uiState                   := 99;
END_IF

CASE uiState OF
  20:
    stState.bBusy           := FALSE;
    eStateActive            := eState + e_AxisFunction.AXIS_DONE;
    eStateExec	            := e_AxisFunction.AXIS_DONE;

  99:
    stState.bError          := TRUE;
    stState.bBusy           := FALSE;

    eStateActive            := eState + e_AxisFunction.ERROR;
    eStateExec	            := e_AxisFunction.ERROR;
END_CASE
END_ACTION

ACTION Axis_Gear_In:
CASE uiState OF
  0:
    eStateActive            := eState;
    stState.bBusy           := TRUE;

    IF (_pAxis1 <> 0)
    THEN
      fbGearIn(Master       := _pAxis1^, 
               Slave        := fbAxis.pAxisRef^, 
               Execute      := FALSE);
 
        uiState             := 10;

    ELSE
      stMsg.eType           := E_MessageType.eMessageError;
      stMsg.eDevice         := e_Device.Axis + TO_INT(fbAxis.pAxisRef^.NcToPlc.AxisId);
      stMsg.eSubdevice      := e_Subdevice.fbGearIn;
      stMsg.iErrorNumber    := 666;
      stMsg.sText           := 'Pointer to Masteraxis null';
      f_MessageSet(stMsg);

      stState.uiErrorId		  := TO_UDINT(stMsg.iErrorNumber);

      uiState               :=99;
    END_IF
    
END_CASE
CASE uiState OF
  10:
    eStateActive            := eState + e_AxisFunction.AXIS_BUSY;
    eStateExec	            := e_AxisFunction.AXIS_BUSY;

    fbGearIn(Master         := _pAxis1^, 
             Slave          := fbAxis.pAxisRef^, 
             Execute        := TRUE,
             RatioNumerator := _stGearIn.RatioNumerator, 
             RatioDenominator:= _stGearIn.RatioDenominator, 
             Acceleration   := _stGearIn.Acceleration, 
             Deceleration   := _stGearIn.Deceleration, 
             Jerk           := _stGearIn.Jerk);

    IF NOT fbGearIn.Error
    THEN
      IF fbGearIn.InGear
      THEN
        fbGearIn(Master     := _pAxis1^, 
                 Slave      := fbAxis._AxisRef, 
                 Execute    := FALSE);

        uiState             := 20;
      END_IF
    ELSE
      stMsg.eType           := E_MessageType.eMessageError;
      stMsg.eDevice         := e_Device.Axis + TO_INT(fbAxis.pAxisRef^.NcToPlc.AxisId);
      stMsg.eSubdevice      := e_Subdevice.fbGearIn;
      stMsg.iErrorNumber    := fbGearIn.ErrorID;
      stMsg.sText           := 'error while gear in';
      f_MessageSet(stMsg);

      stState.uiErrorId		  := TO_UDINT(stMsg.iErrorNumber);

      fbGearIn(Master       := _pAxis1^, 
               Slave        := fbAxis.pAxisRef^, 
               Execute      := FALSE);

      uiState               := 99;
    END_IF
END_CASE
CASE uiState OF
  20:
    stState.bBusy           := FALSE;
    eStateActive            := eState + e_AxisFunction.AXIS_DONE;
    eStateExec	            := e_AxisFunction.AXIS_DONE;

  99:
    stState.bError          := TRUE;
    stState.bBusy           := FALSE;
    eStateActive            := eState + e_AxisFunction.ERROR;
    eStateExec	            := e_AxisFunction.ERROR;
END_CASE
END_ACTION

ACTION Axis_Gear_In_Multimaster:
CASE uiState OF
  0:
    eStateActive                      := eState;
    stState.bBusy                     := TRUE;
    stState.bReady                    := FALSE;

    IF (_pAxis1 <> 0) AND 
       (_pAxis2 <> 0) AND 
       (_pAxis3 <> 0)
    THEN
      fbGearInMultiMaster(Master1     := _pAxis1^,
                          Master2     := _pAxis2^,
                          Master3     := _pAxis3^,
                          Master4     := st_AxisREF_Dummy,//_pAxis4^,
                          Slave       := fbAxis.pAxisRef^,
                          Enable      := FALSE);

      uiState                         := 10;
    ELSE
      stMsg.eType                     := E_MessageType.eMessageError;
      stMsg.eDevice                   := e_Device.Axis + TO_DINT(fbAxis.pAxisRef^.NcToPlc.AxisId);
      stMsg.eSubdevice                := e_Subdevice.fbGearInMultiMaster;
      stMsg.iErrorNumber              := 666;
      stMsg.sText                     := 'Pointer to Master axis null';

      f_MessageSet(stMsg);

      stState.uiErrorId		            := TO_UDINT(stMsg.iErrorNumber);

      uiState                         := 99;
    END_IF
    
END_CASE
CASE uiState OF
  10:
    eStateActive                      := eState + e_AxisFunction.AXIS_BUSY;
    eStateExec	                      := e_AxisFunction.AXIS_BUSY;

    fbGearInMultiMaster(Master1       := _pAxis1^,
                        Master2       := _pAxis2^,
                        Master3       := _pAxis3^,
                        Master4       := st_AxisREF_Dummy,//_pAxis4^,
                        Slave         := fbAxis.pAxisRef^,
                        Enable        := TRUE,
                        GearRatio1    := _stGearInMultiMaster.GearRatio1,
                        GearRatio2    := _stGearInMultiMaster.GearRatio2,
                        GearRatio3    := _stGearInMultiMaster.GearRatio3,
                        GearRatio4    := _stGearInMultiMaster.GearRatio4,
                        Acceleration  := _stGearInMultiMaster.Acceleration, 
                        Deceleration  := _stGearInMultiMaster.Deceleration, 
                        Jerk          := _stGearInMultiMaster.Jerk);

    IF NOT fbGearInMultiMaster.Error
    THEN
      IF fbGearInMultiMaster.InGear
      THEN
        fbGearInMultiMaster(Master1   := _pAxis1^,
                            Master2   := _pAxis2^,
                            Master3   := _pAxis3^,
                            Master4   := st_AxisREF_Dummy,//_pAxis4^,
                            Slave     := fbAxis.pAxisRef^,
                            Enable    := FALSE);

        uiState                       := 20;
      END_IF
    ELSE
      stMsg.eType                     := E_MessageType.eMessageError;
      stMsg.eDevice                   := e_Device.Axis + UDINT_TO_DINT(fbAxis.pAxisRef^.NcToPlc.AxisId);
      stMsg.eSubdevice                := e_Subdevice.fbGearIn;
      stMsg.iErrorNumber              := fbGearIn.ErrorID;
      stMsg.sText                     := 'error while gear in';
      f_MessageSet(stMsg);

      stState.uiErrorId		            := TO_UDINT(stMsg.iErrorNumber);
  
      fbGearInMultiMaster(Master1     := _pAxis1^,
                          Master2     := _pAxis2^,
                          Master3     := _pAxis3^,
                          Master4     := st_AxisREF_Dummy,//_pAxis4^,
                          Slave       := fbAxis.pAxisRef^,
                          Enable      := FALSE);
      uiState := 99;
    END_IF
END_CASE
CASE uiState OF
  20:
    stState.bBusy                     := FALSE;
    eStateActive                      := eState + e_AxisFunction.AXIS_DONE;
    eStateExec	                      := e_AxisFunction.AXIS_DONE;

  99:
    stState.bError                    := TRUE;
    stState.bBusy                     := FALSE;
    eStateActive                      := eState + e_AxisFunction.ERROR;
    eStateExec	                      := e_AxisFunction.ERROR;
END_CASE
END_ACTION

ACTION Axis_Gear_Out:
CASE uiState OF
  0:
    eStateActive            := eState;
    stState.bBusy           := TRUE;

    fbGearOut(Slave         := fbAxis.pAxisRef^, 
              Execute       := FALSE);

    IF NOT fbAxis.pAxisRef^.Status.Coupled
    THEN
      uiState               := 20;
    ELSE
      uiState               := 10;
    END_IF
END_CASE
CASE uiState OF
  10:
    eStateActive            := eState + e_AxisFunction.AXIS_BUSY;
    eStateExec	            := e_AxisFunction.AXIS_BUSY;

    fbGearOut(Slave         := fbAxis.pAxisRef^, 
              Execute       := TRUE);

    IF fbGearOut.Error
    THEN
      stMsg.eType           := E_MessageType.eMessageError;
      stMsg.eDevice         := e_Device.Axis + TO_INT(fbAxis.pAxisRef^.NcToPlc.AxisId);
      stMsg.eSubdevice      := e_Subdevice.fbGearIn;
      stMsg.iErrorNumber    := fbGearOut.ErrorID;
      stMsg.sText           := 'error while gear out';
      f_MessageSet(stMsg);

      stState.uiErrorId		  := TO_UDINT(stMsg.iErrorNumber);

      fbGearOut(Slave       := fbAxis.pAxisRef^, 
                Execute     := FALSE);

      uiState               := 90;

    ELSIF NOT fbAxis.pAxisRef^.Status.Coupled
    THEN
      fbGearOut(Slave       := fbAxis.pAxisRef^, 
                Execute     := FALSE);

